LIN {X 0,Y 408.021,Z 164.665,A -85,B 0,C 180,E1 -11041.457,E2 -11041.457} C_VEL
LIN {X 0,Y 408.969,Z 167.841,A -85,B 0,C 180,E1 -11041.957,E2 -11041.957} C_VEL
LIN {X 0,Y 417.373,Z 186.722,A -85,B 0,C 180,E1 -11042.944,E2 -11042.944} C_VEL
LIN {X 0,Y 418.516,Z 191.213,A -85,B 0,C 180,E1 -11043.111,E2 -11043.111} C_VEL
LIN {X 0,Y 416.527,Z 295.761,A -85,B 0,C 180,E1 -11044.949,E2 -11044.949} C_VEL
LIN {X 0,Y 415.758,Z 335.441,A -85,B 0,C 180,E1 -11045.676,E2 -11045.676} C_VEL
LIN {X 0,Y 415.307,Z 350.191,A -85,B 0,C 180,E1 -11046.129,E2 -11046.129} C_VEL
LIN {X 0,Y 414.66,Z 364.218,A -85,B 0,C 180,E1 -11046.741,E2 -11046.741} C_VEL
LIN {X 0,Y 414.075,Z 373.718,A -85,B 0,C 180,E1 -11047.26,E2 -11047.26} C_VEL
LIN {X 0,Y 413.146,Z 379.141,A -85,B 0,C 180,E1 -11047.557,E2 -11047.557} C_VEL
LIN {X 0,Y 409.846,Z 387.886,A -85,B 0,C 180,E1 -11048.015,E2 -11048.015} C_VEL
LIN {X 0,Y 406.373,Z 396.437,A -85,B 0,C 180,E1 -11048.54,E2 -11048.54} C_VEL
LIN {X 0,Y 405.151,Z 401.412,A -85,B 0,C 180,E1 -11048.948,E2 -11048.948} C_VEL
LIN {X 0,Y 403.781,Z 413.481,A -85,B 0,C 180,E1 -11050.194,E2 -11050.194} C_VEL
LIN {X 0,Y 402.539,Z 425.332,A -85,B 0,C 180,E1 -11051.682,E2 -11051.682} C_VEL
LIN {X 0,Y 401.227,Z 435.48,A -85,B 0,C 180,E1 -11053.2,E2 -11053.2} C_VEL
LIN {X 0,Y 399.908,Z 445.382,A -85,B 0,C 180,E1 -11054.975,E2 -11054.975} C_VEL
LIN {X 0,Y 398.903,Z 453.589,A -85,B 0,C 180,E1 -11056.758,E2 -11056.758} C_VEL
LIN {X 0,Y 397.976,Z 461.263,A -85,B 0,C 180,E1 -11058.798,E2 -11058.798} C_VEL
LIN {X 0,Y 397.275,Z 467.361,A -85,B 0,C 180,E1 -11060.837,E2 -11060.837} C_VEL
LIN {X 0,Y 396.768,Z 472.074,A -85,B 0,C 180,E1 -11062.876,E2 -11062.876} C_VEL
LIN {X 0,Y 396.541,Z 475.518,A -85,B 0,C 180,E1 -11064.915,E2 -11064.915} C_VEL
LIN {X 0,Y 396.369,Z 477.793,A -85,B 0,C 180,E1 -11066.95,E2 -11066.95} C_VEL
LIN {X 0,Y 396.082,Z 478.967,A -85,B 0,C 180,E1 -11068.982,E2 -11068.982} C_VEL
LIN {X 0,Y 396.081,Z 478.981,A -85,B 0,C 180,E1 -11071.015,E2 -11071.015} C_VEL
LIN {X 0,Y 396.367,Z 477.865,A -85,B 0,C 180,E1 -11073.048,E2 -11073.048} C_VEL
LIN {X 0,Y 396.529,Z 475.652,A -85,B 0,C 180,E1 -11075.083,E2 -11075.083} C_VEL
LIN {X 0,Y 396.764,Z 472.277,A -85,B 0,C 180,E1 -11077.121,E2 -11077.121} C_VEL
LIN {X 0,Y 397.269,Z 467.633,A -85,B 0,C 180,E1 -11079.16,E2 -11079.16} C_VEL
LIN {X 0,Y 397.952,Z 461.602,A -85,B 0,C 180,E1 -11081.2,E2 -11081.2} C_VEL
LIN {X 0,Y 398.867,Z 454.005,A -85,B 0,C 180,E1 -11083.24,E2 -11083.24} C_VEL
LIN {X 0,Y 399.845,Z 445.978,A -85,B 0,C 180,E1 -11085.008,E2 -11085.008} C_VEL
LIN {X 0,Y 401.166,Z 436.091,A -85,B 0,C 180,E1 -11086.8,E2 -11086.8} C_VEL
LIN {X 0,Y 402.459,Z 426.066,A -85,B 0,C 180,E1 -11088.319,E2 -11088.319} C_VEL
LIN {X 0,Y 403.698,Z 414.655,A -85,B 0,C 180,E1 -11089.773,E2 -11089.773} C_VEL
LIN {X 0,Y 405.129,Z 402.003,A -85,B 0,C 180,E1 -11091.096,E2 -11091.096} C_VEL
LIN {X 0,Y 406.489,Z 388.828,A -85,B 0,C 180,E1 -11092.221,E2 -11092.221} C_VEL
LIN {X 0,Y 407.563,Z 375.261,A -85,B 0,C 180,E1 -11093.163,E2 -11093.163} C_VEL
LIN {X 0,Y 408.376,Z 361.756,A -85,B 0,C 180,E1 -11093.904,E2 -11093.904} C_VEL
LIN {X 0,Y 409.06,Z 346.686,A -85,B 0,C 180,E1 -11094.519,E2 -11094.519} C_VEL
LIN {X 0,Y 409.496,Z 331.535,A -85,B 0,C 180,E1 -11094.931,E2 -11094.931} C_VEL
LIN {X 0,Y 412.244,Z 193.174,A -85,B 0,C 180,E1 -11097.405,E2 -11097.405} C_VEL
LIN {X 0,Y 411.218,Z 189.005,A -85,B 0,C 180,E1 -11097.561,E2 -11097.561} C_VEL
LIN {X 0,Y 402.554,Z 169.768,A -85,B 0,C 180,E1 -11098.604,E2 -11098.604} C_VEL
LIN {X 0,Y 401.881,Z 168.212,A -85,B 0,C 180,E1 -11098.709,E2 -11098.709} C_VEL
LIN {X 0,Y 397.118,Z 152.67,A -85,B 0,C 180,E1 -11101.396,E2 -11101.396} C_VEL
LIN {X 0,Y 397.121,Z 152.643,A -85,B 0,C 180,E1 -11104.492,E2 -11104.492} C_VEL
LIN {X 0,Y 397.098,Z 152.644,A -85,B 0,C 180,E1 -11108.273,E2 -11108.273} C_VEL
LIN {X 0,Y 397.085,Z 152.629,A -85,B 0,C 180,E1 -11110.907,E2 -11110.907} C_VEL
LIN {X 0,Y 397.098,Z 152.641,A -85,B 0,C 180,E1 -11113.647,E2 -11113.647} C_VEL
LIN {X 0,Y 397.097,Z 152.645,A -85,B 0,C 180,E1 -11116.519,E2 -11116.519} C_VEL
LIN {X 0,Y 397.113,Z 152.644,A -85,B 0,C 180,E1 -11119.55,E2 -11119.55} C_VEL
LIN {X 0,Y 397.091,Z 152.645,A -85,B 0,C 180,E1 -11122.789,E2 -11122.789} C_VEL
LIN {X 0,Y 397.11,Z 152.637,A -85,B 0,C 180,E1 -11126.281,E2 -11126.281} C_VEL
LIN {X 0,Y 397.079,Z 152.64,A -85,B 0,C 180,E1 -11129.117,E2 -11129.117} C_VEL
LIN {X 0,Y 397.185,Z 152.635,A -85,B 0,C 180,E1 -11132.609,E2 -11132.609} C_VEL
LIN {X 0,Y 397.119,Z 152.633,A -85,B 0,C 180,E1 -11135.981,E2 -11135.981} C_VEL
LIN {X 0,Y 397.128,Z 152.633,A -85,B 0,C 180,E1 -11139.704,E2 -11139.704} C_VEL
LIN {X 0,Y 397.171,Z 152.633,A -85,B 0,C 180,E1 -11142.844,E2 -11142.844} C_VEL
LIN {X 0,Y 397.215,Z 152.617,A -85,B 0,C 180,E1 -11146.678,E2 -11146.678} C_VEL
LIN {X 0,Y 397.208,Z 152.629,A -85,B 0,C 180,E1 -11149.809,E2 -11149.809} C_VEL
LIN {X 0,Y 397.353,Z 152.598,A -85,B 0,C 180,E1 -11152.888,E2 -11152.888} C_VEL
LIN {X 0,Y 397.245,Z 152.619,A -85,B 0,C 180,E1 -11154.925,E2 -11154.925} C_VEL
LIN {X 0,Y 397.441,Z 152.6,A -85,B 0,C 180,E1 -11157.973,E2 -11157.973} C_VEL
LIN {X 0,Y 397.571,Z 152.569,A -85,B 0,C 180,E1 -11160,E2 -11160} C_VEL
LIN {X 0,Y 397.372,Z 152.611,A -85,B 0,C 180,E1 -11163.041,E2 -11163.041} C_VEL
LIN {X 0,Y 397.352,Z 152.597,A -85,B 0,C 180,E1 -11167.112,E2 -11167.112} C_VEL
LIN {X 0,Y 397.208,Z 152.629,A -85,B 0,C 180,E1 -11170.191,E2 -11170.191} C_VEL
LIN {X 0,Y 397.215,Z 152.613,A -85,B 0,C 180,E1 -11173.321,E2 -11173.321} C_VEL
LIN {X 0,Y 397.16,Z 152.637,A -85,B 0,C 180,E1 -11176.447,E2 -11176.447} C_VEL
LIN {X 0,Y 397.137,Z 152.625,A -85,B 0,C 180,E1 -11179.648,E2 -11179.648} C_VEL
LIN {X 0,Y 397.125,Z 152.635,A -85,B 0,C 180,E1 -11183.041,E2 -11183.041} C_VEL
LIN {X 0,Y 397.125,Z 152.639,A -85,B 0,C 180,E1 -11186.259,E2 -11186.259} C_VEL
LIN {X 0,Y 397.111,Z 152.637,A -85,B 0,C 180,E1 -11188.544,E2 -11188.544} C_VEL
LIN {X 0,Y 397.069,Z 152.651,A -85,B 0,C 180,E1 -11192.072,E2 -11192.072} C_VEL
LIN {X 0,Y 397.11,Z 152.64,A -85,B 0,C 180,E1 -11195.504,E2 -11195.504} C_VEL
LIN {X 0,Y 397.123,Z 152.623,A -85,B 0,C 180,E1 -11198.863,E2 -11198.863} C_VEL
LIN {X 0,Y 397.059,Z 152.636,A -85,B 0,C 180,E1 -11202.268,E2 -11202.268} C_VEL
LIN {X 0,Y 397.109,Z 152.643,A -85,B 0,C 180,E1 -11205.065,E2 -11205.065} C_VEL
LIN {X 0,Y 397.149,Z 152.642,A -85,B 0,C 180,E1 -11208.008,E2 -11208.008} C_VEL
LIN {X 0,Y 397.135,Z 152.637,A -85,B 0,C 180,E1 -11211.989,E2 -11211.989} C_VEL
LIN {X 0,Y 403.812,Z 174.916,A -85,B 0,C 180,E1 -11215.514,E2 -11215.514} C_VEL
LIN {X 0,Y 408.122,Z 189.921,A -85,B 0,C 180,E1 -11217.737,E2 -11217.737} C_VEL
LIN {X 0,Y 405.393,Z 216.791,A -85,B 0,C 180,E1 -11220.962,E2 -11220.962} C_VEL
LIN {X 0,Y 404.786,Z 223.542,A -85,B 0,C 180,E1 -11221.752,E2 -11221.752} C_VEL
LIN {X 0,Y 410.254,Z 268.107,A -85,B 0,C 180,E1 -11223.009,E2 -11223.009} C_VEL
LIN {X 0,Y 408.286,Z 377.569,A -85,B 0,C 180,E1 -11224.956,E2 -11224.956} C_VEL
LIN {X 0,Y 407.723,Z 400.403,A -85,B 0,C 180,E1 -11225.395,E2 -11225.395} C_VEL
LIN {X 0,Y 406.837,Z 415.914,A -85,B 0,C 180,E1 -11225.881,E2 -11225.881} C_VEL
LIN {X 0,Y 405.754,Z 430.277,A -85,B 0,C 180,E1 -11226.525,E2 -11226.525} C_VEL
LIN {X 0,Y 404.634,Z 443.502,A -85,B 0,C 180,E1 -11227.304,E2 -11227.304} C_VEL
LIN {X 0,Y 403.02,Z 458.122,A -85,B 0,C 180,E1 -11228.386,E2 -11228.386} C_VEL
LIN {X 0,Y 401.573,Z 471.663,A -85,B 0,C 180,E1 -11229.647,E2 -11229.647} C_VEL
LIN {X 0,Y 400.174,Z 483.977,A -85,B 0,C 180,E1 -11231.042,E2 -11231.042} C_VEL
LIN {X 0,Y 398.967,Z 495.231,A -85,B 0,C 180,E1 -11232.576,E2 -11232.576} C_VEL
LIN {X 0,Y 397.956,Z 504.72,A -85,B 0,C 180,E1 -11234.115,E2 -11234.115} C_VEL
LIN {X 0,Y 397.129,Z 514.055,A -85,B 0,C 180,E1 -11235.918,E2 -11235.918} C_VEL
LIN {X 0,Y 396.519,Z 521.815,A -85,B 0,C 180,E1 -11237.721,E2 -11237.721} C_VEL
LIN {X 0,Y 396.257,Z 527.426,A -85,B 0,C 180,E1 -11239.269,E2 -11239.269} C_VEL
LIN {X 0,Y 396.049,Z 533.524,A -85,B 0,C 180,E1 -11241.326,E2 -11241.326} C_VEL
LIN {X 0,Y 396.1,Z 538.462,A -85,B 0,C 180,E1 -11243.517,E2 -11243.517} C_VEL
LIN {X 0,Y 396.103,Z 540.808,A -85,B 0,C 180,E1 -11244.912,E2 -11244.912} C_VEL
LIN {X 0,Y 396.218,Z 543.231,A -85,B 0,C 180,E1 -11246.951,E2 -11246.951} C_VEL
LIN {X 0,Y 396.217,Z 544.445,A -85,B 0,C 180,E1 -11248.985,E2 -11248.985} C_VEL
LIN {X 0,Y 396.204,Z 544.443,A -85,B 0,C 180,E1 -11251.018,E2 -11251.018} C_VEL
LIN {X 0,Y 396.219,Z 543.229,A -85,B 0,C 180,E1 -11253.052,E2 -11253.052} C_VEL
LIN {X 0,Y 396.098,Z 540.8,A -85,B 0,C 180,E1 -11255.091,E2 -11255.091} C_VEL
LIN {X 0,Y 396.093,Z 537.12,A -85,B 0,C 180,E1 -11257.136,E2 -11257.136} C_VEL
LIN {X 0,Y 396.105,Z 532.099,A -85,B 0,C 180,E1 -11259.19,E2 -11259.19} C_VEL
LIN {X 0,Y 396.378,Z 525.628,A -85,B 0,C 180,E1 -11261.248,E2 -11261.248} C_VEL
LIN {X 0,Y 396.876,Z 517.511,A -85,B 0,C 180,E1 -11263.31,E2 -11263.31} C_VEL
LIN {X 0,Y 397.589,Z 508.865,A -85,B 0,C 180,E1 -11265.115,E2 -11265.115} C_VEL
LIN {X 0,Y 398.671,Z 498.474,A -85,B 0,C 180,E1 -11266.911,E2 -11266.911} C_VEL
LIN {X 0,Y 399.779,Z 487.843,A -85,B 0,C 180,E1 -11268.449,E2 -11268.449} C_VEL
LIN {X 0,Y 401.029,Z 476.284,A -85,B 0,C 180,E1 -11269.85,E2 -11269.85} C_VEL
LIN {X 0,Y 402.443,Z 463.734,A -85,B 0,C 180,E1 -11271.112,E2 -11271.112} C_VEL
LIN {X 0,Y 403.793,Z 451.687,A -85,B 0,C 180,E1 -11272.111,E2 -11272.111} C_VEL
LIN {X 0,Y 405.091,Z 437.85,A -85,B 0,C 180,E1 -11273.043,E2 -11273.043} C_VEL
LIN {X 0,Y 406.35,Z 422.379,A -85,B 0,C 180,E1 -11273.847,E2 -11273.847} C_VEL
LIN {X 0,Y 407.447,Z 406.722,A -85,B 0,C 180,E1 -11274.422,E2 -11274.422} C_VEL
LIN {X 0,Y 407.975,Z 391.263,A -85,B 0,C 180,E1 -11274.795,E2 -11274.795} C_VEL
LIN {X 0,Y 409.35,Z 324.517,A -85,B 0,C 180,E1 -11275.999,E2 -11275.999} C_VEL
LIN {X 0,Y 411.902,Z 267.787,A -85,B 0,C 180,E1 -11277.413,E2 -11277.413} C_VEL
LIN {X 0,Y 410.199,Z 247.528,A -85,B 0,C 180,E1 -11278.216,E2 -11278.216} C_VEL
LIN {X 0,Y 408.178,Z 233.394,A -85,B 0,C 180,E1 -11278.894,E2 -11278.894} C_VEL
LIN {X 0,Y 412.028,Z 211.405,A -85,B 0,C 180,E1 -11281.923,E2 -11281.923} C_VEL
LIN {X 0,Y 414.392,Z 200.57,A -85,B 0,C 180,E1 -11283.492,E2 -11283.492} C_VEL
LIN {X 0,Y 414.398,Z 198.896,A -85,B 0,C 180,E1 -11283.797,E2 -11283.797} C_VEL
LIN {X 0,Y 412.326,Z 190.433,A -85,B 0,C 180,E1 -11285.794,E2 -11285.794} C_VEL
LIN {X 0,Y 409.948,Z 183.181,A -85,B 0,C 180,E1 -11287.945,E2 -11287.945} C_VEL
LIN {X 0,Y 408.411,Z 178.732,A -85,B 0,C 180,E1 -11289.548,E2 -11289.548} C_VEL
LIN {X 0,Y 407.187,Z 175.487,A -85,B 0,C 180,E1 -11290.987,E2 -11290.987} C_VEL
LIN {X 0,Y 405.558,Z 171.699,A -85,B 0,C 180,E1 -11293.296,E2 -11293.296} C_VEL
LIN {X 0,Y 404.597,Z 169.529,A -85,B 0,C 180,E1 -11295.414,E2 -11295.414} C_VEL
LIN {X 0,Y 404.292,Z 168.538,A -85,B 0,C 180,E1 -11297.316,E2 -11297.316} C_VEL
LIN {X 0,Y 404.141,Z 168.532,A -85,B 0,C 180,E1 -11298.638,E2 -11298.638} C_VEL
LIN {X 0,Y 404.304,Z 169.873,A -85,B 0,C 180,E1 -11301.26,E2 -11301.26} C_VEL
LIN {X 0,Y 405.298,Z 172.634,A -85,B 0,C 180,E1 -11303.874,E2 -11303.874} C_VEL
LIN {X 0,Y 406.441,Z 176.266,A -85,B 0,C 180,E1 -11306.1,E2 -11306.1} C_VEL
LIN {X 0,Y 407.654,Z 180.67,A -85,B 0,C 180,E1 -11308.189,E2 -11308.189} C_VEL
LIN {X 0,Y 409.124,Z 187.192,A -85,B 0,C 180,E1 -11310.688,E2 -11310.688} C_VEL
LIN {X 0,Y 410.116,Z 192.489,A -85,B 0,C 180,E1 -11312.439,E2 -11312.439} C_VEL
LIN {X 0,Y 410.527,Z 196.337,A -85,B 0,C 180,E1 -11313.57,E2 -11313.57} C_VEL
LIN {X 0,Y 408.558,Z 207.239,A -85,B 0,C 180,E1 -11316.061,E2 -11316.061} C_VEL
LIN {X 0,Y 408.206,Z 209.863,A -85,B 0,C 180,E1 -11316.608,E2 -11316.608} C_VEL
LIN {X 0,Y 412.045,Z 224.419,A -85,B 0,C 180,E1 -11317.661,E2 -11317.661} C_VEL
LIN {X 0,Y 413.131,Z 229.704,A -85,B 0,C 180,E1 -11317.992,E2 -11317.992} C_VEL
LIN {X 0,Y 407.346,Z 316.237,A -85,B 0,C 180,E1 -11320.668,E2 -11320.668} C_VEL
LIN {X 0,Y 406.778,Z 332.313,A -85,B 0,C 180,E1 -11321.229,E2 -11321.229} C_VEL
LIN {X 0,Y 406.107,Z 346.202,A -85,B 0,C 180,E1 -11321.914,E2 -11321.914} C_VEL
LIN {X 0,Y 405.155,Z 360.459,A -85,B 0,C 180,E1 -11322.849,E2 -11322.849} C_VEL
LIN {X 0,Y 404.107,Z 373.535,A -85,B 0,C 180,E1 -11323.973,E2 -11323.973} C_VEL
LIN {X 0,Y 403.231,Z 384.092,A -85,B 0,C 180,E1 -11325.103,E2 -11325.103} C_VEL
LIN {X 0,Y 402.315,Z 393.688,A -85,B 0,C 180,E1 -11326.36,E2 -11326.36} C_VEL
LIN {X 0,Y 401.261,Z 403.094,A -85,B 0,C 180,E1 -11327.867,E2 -11327.867} C_VEL
LIN {X 0,Y 400.302,Z 411.148,A -85,B 0,C 180,E1 -11329.48,E2 -11329.48} C_VEL
LIN {X 0,Y 399.468,Z 416.812,A -85,B 0,C 180,E1 -11330.89,E2 -11330.89} C_VEL
LIN {X 0,Y 398.948,Z 421.58,A -85,B 0,C 180,E1 -11332.408,E2 -11332.408} C_VEL
LIN {X 0,Y 398.318,Z 425.26,A -85,B 0,C 180,E1 -11333.923,E2 -11333.923} C_VEL
LIN {X 0,Y 398.058,Z 427.078,A -85,B 0,C 180,E1 -11334.936,E2 -11334.936} C_VEL
LIN {X 0,Y 397.873,Z 428.461,A -85,B 0,C 180,E1 -11335.948,E2 -11335.948} C_VEL
LIN {X 0,Y 397.665,Z 429.44,A -85,B 0,C 180,E1 -11336.961,E2 -11336.961} C_VEL
LIN {X 0,Y 397.525,Z 429.977,A -85,B 0,C 180,E1 -11337.974,E2 -11337.974} C_VEL
LIN {X 0,Y 397.299,Z 430.089,A -85,B 0,C 180,E1 -11338.987,E2 -11338.987} C_VEL
LIN {X 0,Y 397.206,Z 429.774,A -85,B 0,C 180,E1 -11340,E2 -11340} C_VEL
LIN {X 0,Y 397.219,Z 429.042,A -85,B 0,C 180,E1 -11341.014,E2 -11341.014} C_VEL
LIN {X 0,Y 397.141,Z 427.889,A -85,B 0,C 180,E1 -11342.028,E2 -11342.028} C_VEL
LIN {X 0,Y 397.147,Z 425.347,A -85,B 0,C 180,E1 -11343.551,E2 -11343.551} C_VEL
LIN {X 0,Y 397.263,Z 421.771,A -85,B 0,C 180,E1 -11345.075,E2 -11345.075} C_VEL
LIN {X 0,Y 397.527,Z 417.087,A -85,B 0,C 180,E1 -11346.599,E2 -11346.599} C_VEL
LIN {X 0,Y 397.823,Z 411.176,A -85,B 0,C 180,E1 -11348.125,E2 -11348.125} C_VEL
LIN {X 0,Y 398.204,Z 403.848,A -85,B 0,C 180,E1 -11349.652,E2 -11349.652} C_VEL
LIN {X 0,Y 398.702,Z 394.845,A -85,B 0,C 180,E1 -11351.181,E2 -11351.181} C_VEL
LIN {X 0,Y 399.232,Z 384.652,A -85,B 0,C 180,E1 -11352.583,E2 -11352.583} C_VEL
LIN {X 0,Y 399.846,Z 373.252,A -85,B 0,C 180,E1 -11353.856,E2 -11353.856} C_VEL
LIN {X 0,Y 400.359,Z 361.658,A -85,B 0,C 180,E1 -11354.907,E2 -11354.907} C_VEL
LIN {X 0,Y 400.866,Z 348.717,A -85,B 0,C 180,E1 -11355.834,E2 -11355.834} C_VEL
LIN {X 0,Y 401.238,Z 336.062,A -85,B 0,C 180,E1 -11356.537,E2 -11356.537} C_VEL
LIN {X 0,Y 401.582,Z 323.646,A -85,B 0,C 180,E1 -11357.046,E2 -11357.046} C_VEL
LIN {X 0,Y 401.849,Z 305.487,A -85,B 0,C 180,E1 -11357.526,E2 -11357.526} C_VEL
LIN {X 0,Y 403.894,Z 221.695,A -85,B 0,C 180,E1 -11359.463,E2 -11359.463} C_VEL
LIN {X 0,Y 400.491,Z 201.256,A -85,B 0,C 180,E1 -11360.141,E2 -11360.141} C_VEL
LIN {X 0,Y 401.81,Z 182.13,A -85,B 0,C 180,E1 -11363.722,E2 -11363.722} C_VEL
LIN {X 0,Y 402.035,Z 175.04,A -85,B 0,C 180,E1 -11365.082,E2 -11365.082} C_VEL
LIN {X 0,Y 399.379,Z 162.271,A -85,B 0,C 180,E1 -11367.757,E2 -11367.757} C_VEL
LIN {X 0,Y 397.107,Z 152.647,A -85,B 0,C 180,E1 -11369.863,E2 -11369.863} C_VEL
LIN {X 0,Y 397.124,Z 152.644,A -85,B 0,C 180,E1 -11373.717,E2 -11373.717} C_VEL
LIN {X 0,Y 397.097,Z 152.648,A -85,B 0,C 180,E1 -11377.208,E2 -11377.208} C_VEL
LIN {X 0,Y 397.082,Z 152.639,A -85,B 0,C 180,E1 -11380.441,E2 -11380.441} C_VEL
LIN {X 0,Y 397.105,Z 152.637,A -85,B 0,C 180,E1 -11383.648,E2 -11383.648} C_VEL
LIN {X 0,Y 397.107,Z 152.643,A -85,B 0,C 180,E1 -11386.52,E2 -11386.52} C_VEL
LIN {X 0,Y 397.118,Z 152.639,A -85,B 0,C 180,E1 -11390.422,E2 -11390.422} C_VEL
LIN {X 0,Y 397.112,Z 152.649,A -85,B 0,C 180,E1 -11394.265,E2 -11394.265} C_VEL
LIN {X 0,Y 397.119,Z 152.644,A -85,B 0,C 180,E1 -11396.726,E2 -11396.726} C_VEL
LIN {X 0,Y 397.125,Z 152.734,A -85,B 0,C 180,E1 -11398.713,E2 -11398.713} C_VEL
LIN {X 0,Y 401.677,Z 167.617,A -85,B 0,C 180,E1 -11401.3,E2 -11401.3} C_VEL
LIN {X 0,Y 401.981,Z 168.544,A -85,B 0,C 180,E1 -11401.429,E2 -11401.429} C_VEL
LIN {X 0,Y 410.806,Z 187.932,A -85,B 0,C 180,E1 -11402.488,E2 -11402.488} C_VEL
LIN {X 0,Y 412.127,Z 192.143,A -85,B 0,C 180,E1 -11402.668,E2 -11402.668} C_VEL
LIN {X 0,Y 410.317,Z 287.367,A -85,B 0,C 180,E1 -11404.373,E2 -11404.373} C_VEL
LIN {X 0,Y 409.324,Z 335.96,A -85,B 0,C 180,E1 -11405.268,E2 -11405.268} C_VEL
LIN {X 0,Y 408.852,Z 350.887,A -85,B 0,C 180,E1 -11405.734,E2 -11405.734} C_VEL
LIN {X 0,Y 408.173,Z 364.968,A -85,B 0,C 180,E1 -11406.36,E2 -11406.36} C_VEL
LIN {X 0,Y 407.292,Z 378.606,A -85,B 0,C 180,E1 -11407.153,E2 -11407.153} C_VEL
LIN {X 0,Y 406.113,Z 392.307,A -85,B 0,C 180,E1 -11408.156,E2 -11408.156} C_VEL
LIN {X 0,Y 405.151,Z 401.412,A -85,B 0,C 180,E1 -11408.948,E2 -11408.948} C_VEL
LIN {X 0,Y 403.955,Z 406.344,A -85,B 0,C 180,E1 -11409.378,E2 -11409.378} C_VEL
LIN {X 0,Y 400.447,Z 414.245,A -85,B 0,C 180,E1 -11410.068,E2 -11410.068} C_VEL
LIN {X 0,Y 396.954,Z 421.797,A -85,B 0,C 180,E1 -11410.839,E2 -11410.839} C_VEL
LIN {X 0,Y 395.793,Z 426.121,A -85,B 0,C 180,E1 -11411.389,E2 -11411.389} C_VEL
LIN {X 0,Y 394.451,Z 436.062,A -85,B 0,C 180,E1 -11412.902,E2 -11412.902} C_VEL
LIN {X 0,Y 393.089,Z 445.755,A -85,B 0,C 180,E1 -11414.665,E2 -11414.665} C_VEL
LIN {X 0,Y 392.014,Z 454.174,A -85,B 0,C 180,E1 -11416.521,E2 -11416.521} C_VEL
LIN {X 0,Y 391.009,Z 461.85,A -85,B 0,C 180,E1 -11418.595,E2 -11418.595} C_VEL
LIN {X 0,Y 390.274,Z 467.948,A -85,B 0,C 180,E1 -11420.672,E2 -11420.672} C_VEL
LIN {X 0,Y 389.748,Z 472.659,A -85,B 0,C 180,E1 -11422.747,E2 -11422.747} C_VEL
LIN {X 0,Y 389.485,Z 476.104,A -85,B 0,C 180,E1 -11424.822,E2 -11424.822} C_VEL
LIN {X 0,Y 389.298,Z 478.379,A -85,B 0,C 180,E1 -11426.894,E2 -11426.894} C_VEL
LIN {X 0,Y 389.031,Z 479.55,A -85,B 0,C 180,E1 -11428.964,E2 -11428.964} C_VEL
LIN {X 0,Y 389.03,Z 479.564,A -85,B 0,C 180,E1 -11431.034,E2 -11431.034} C_VEL
LIN {X 0,Y 389.296,Z 478.45,A -85,B 0,C 180,E1 -11433.103,E2 -11433.103} C_VEL
LIN {X 0,Y 389.473,Z 476.237,A -85,B 0,C 180,E1 -11435.175,E2 -11435.175} C_VEL
LIN {X 0,Y 389.804,Z 472.524,A -85,B 0,C 180,E1 -11437.419,E2 -11437.419} C_VEL
LIN {X 0,Y 390.267,Z 468.217,A -85,B 0,C 180,E1 -11439.326,E2 -11439.326} C_VEL
LIN {X 0,Y 390.982,Z 462.186,A -85,B 0,C 180,E1 -11441.403,E2 -11441.403} C_VEL
LIN {X 0,Y 391.979,Z 454.585,A -85,B 0,C 180,E1 -11443.477,E2 -11443.477} C_VEL
LIN {X 0,Y 393,Z 446.678,A -85,B 0,C 180,E1 -11445.251,E2 -11445.251} C_VEL
LIN {X 0,Y 394.183,Z 438.211,A -85,B 0,C 180,E1 -11446.84,E2 -11446.84} C_VEL
LIN {X 0,Y 395.503,Z 428.421,A -85,B 0,C 180,E1 -11448.384,E2 -11448.384} C_VEL
LIN {X 0,Y 396.863,Z 417.195,A -85,B 0,C 180,E1 -11449.876,E2 -11449.876} C_VEL
LIN {X 0,Y 398.228,Z 405.136,A -85,B 0,C 180,E1 -11451.208,E2 -11451.208} C_VEL
LIN {X 0,Y 399.617,Z 392.51,A -85,B 0,C 180,E1 -11452.352,E2 -11452.352} C_VEL
LIN {X 0,Y 400.802,Z 378.716,A -85,B 0,C 180,E1 -11453.372,E2 -11453.372} C_VEL
LIN {X 0,Y 401.83,Z 364.343,A -85,B 0,C 180,E1 -11454.204,E2 -11454.204} C_VEL
LIN {X 0,Y 402.491,Z 349.785,A -85,B 0,C 180,E1 -11454.843,E2 -11454.843} C_VEL
LIN {X 0,Y 402.995,Z 334.732,A -85,B 0,C 180,E1 -11455.293,E2 -11455.293} C_VEL
LIN {X 0,Y 405.875,Z 198.835,A -85,B 0,C 180,E1 -11457.769,E2 -11457.769} C_VEL
LIN {X 0,Y 405.868,Z 193.622,A -85,B 0,C 180,E1 -11457.872,E2 -11457.872} C_VEL
LIN {X 0,Y 400.034,Z 179.778,A -85,B 0,C 180,E1 -11458.603,E2 -11458.603} C_VEL
LIN {X 0,Y 394.796,Z 168.752,A -85,B 0,C 180,E1 -11459.275,E2 -11459.275} C_VEL
LIN {X 0,Y 390.908,Z 156.366,A -85,B 0,C 180,E1 -11461.423,E2 -11461.423} C_VEL
LIN {X 0,Y 390.04,Z 153.515,A -85,B 0,C 180,E1 -11461.987,E2 -11461.987} C_VEL
LIN {X 0,Y 390.081,Z 153.521,A -85,B 0,C 180,E1 -11465.205,E2 -11465.205} C_VEL
LIN {X 0,Y 390.084,Z 153.505,A -85,B 0,C 180,E1 -11469.091,E2 -11469.091} C_VEL
LIN {X 0,Y 390.057,Z 153.522,A -85,B 0,C 180,E1 -11472.376,E2 -11472.376} C_VEL
LIN {X 0,Y 390.048,Z 153.523,A -85,B 0,C 180,E1 -11476.112,E2 -11476.112} C_VEL
LIN {X 0,Y 390.067,Z 153.521,A -85,B 0,C 180,E1 -11479.562,E2 -11479.562} C_VEL
LIN {X 0,Y 390.039,Z 153.521,A -85,B 0,C 180,E1 -11482.447,E2 -11482.447} C_VEL
LIN {X 0,Y 390.075,Z 153.514,A -85,B 0,C 180,E1 -11486.046,E2 -11486.046} C_VEL
LIN {X 0,Y 390.036,Z 153.511,A -85,B 0,C 180,E1 -11489.7,E2 -11489.7} C_VEL
LIN {X 0,Y 390.104,Z 153.516,A -85,B 0,C 180,E1 -11493.231,E2 -11493.231} C_VEL
LIN {X 0,Y 390.066,Z 153.516,A -85,B 0,C 180,E1 -11496.76,E2 -11496.76} C_VEL
LIN {X 0,Y 390.093,Z 153.509,A -85,B 0,C 180,E1 -11499.982,E2 -11499.982} C_VEL
LIN {X 0,Y 390.127,Z 153.515,A -85,B 0,C 180,E1 -11503.248,E2 -11503.248} C_VEL
LIN {X 0,Y 390.183,Z 153.494,A -85,B 0,C 180,E1 -11506.561,E2 -11506.561} C_VEL
LIN {X 0,Y 390.159,Z 153.508,A -85,B 0,C 180,E1 -11509.622,E2 -11509.622} C_VEL
LIN {X 0,Y 390.307,Z 153.477,A -85,B 0,C 180,E1 -11512.759,E2 -11512.759} C_VEL
LIN {X 0,Y 390.217,Z 153.492,A -85,B 0,C 180,E1 -11514.833,E2 -11514.833} C_VEL
LIN {X 0,Y 390.41,Z 153.476,A -85,B 0,C 180,E1 -11517.937,E2 -11517.937} C_VEL
LIN {X 0,Y 390.541,Z 153.444,A -85,B 0,C 180,E1 -11520,E2 -11520} C_VEL
LIN {X 0,Y 390.306,Z 153.49,A -85,B 0,C 180,E1 -11523.096,E2 -11523.096} C_VEL
LIN {X 0,Y 390.319,Z 153.474,A -85,B 0,C 180,E1 -11526.202,E2 -11526.202} C_VEL
LIN {X 0,Y 390.303,Z 153.48,A -85,B 0,C 180,E1 -11528.282,E2 -11528.282} C_VEL
LIN {X 0,Y 390.16,Z 153.493,A -85,B 0,C 180,E1 -11532.483,E2 -11532.483} C_VEL
LIN {X 0,Y 390.133,Z 153.507,A -85,B 0,C 180,E1 -11535.677,E2 -11535.677} C_VEL
LIN {X 0,Y 390.095,Z 153.501,A -85,B 0,C 180,E1 -11538.922,E2 -11538.922} C_VEL
LIN {X 0,Y 390.031,Z 153.527,A -85,B 0,C 180,E1 -11542.235,E2 -11542.235} C_VEL
LIN {X 0,Y 390.108,Z 153.508,A -85,B 0,C 180,E1 -11545.744,E2 -11545.744} C_VEL
LIN {X 0,Y 390.048,Z 153.512,A -85,B 0,C 180,E1 -11549.11,E2 -11549.11} C_VEL
LIN {X 0,Y 390.033,Z 153.523,A -85,B 0,C 180,E1 -11552.722,E2 -11552.722} C_VEL
LIN {X 0,Y 390.048,Z 153.522,A -85,B 0,C 180,E1 -11555.827,E2 -11555.827} C_VEL
LIN {X 0,Y 390.062,Z 153.495,A -85,B 0,C 180,E1 -11559.22,E2 -11559.22} C_VEL
LIN {X 0,Y 390.033,Z 153.513,A -85,B 0,C 180,E1 -11562.375,E2 -11562.375} C_VEL
LIN {X 0,Y 390.098,Z 153.519,A -85,B 0,C 180,E1 -11566.107,E2 -11566.107} C_VEL
LIN {X 0,Y 390.075,Z 153.521,A -85,B 0,C 180,E1 -11569.175,E2 -11569.175} C_VEL
LIN {X 0,Y 390.093,Z 153.561,A -85,B 0,C 180,E1 -11571.564,E2 -11571.564} C_VEL
LIN {X 0,Y 396.406,Z 174.706,A -85,B 0,C 180,E1 -11574.967,E2 -11574.967} C_VEL
LIN {X 0,Y 401.15,Z 191.216,A -85,B 0,C 180,E1 -11577.472,E2 -11577.472} C_VEL
LIN {X 0,Y 401.189,Z 193.586,A -85,B 0,C 180,E1 -11577.783,E2 -11577.783} C_VEL
LIN {X 0,Y 398.167,Z 221.719,A -85,B 0,C 180,E1 -11581.209,E2 -11581.209} C_VEL
LIN {X 0,Y 403.756,Z 267.493,A -85,B 0,C 180,E1 -11582.535,E2 -11582.535} C_VEL
LIN {X 0,Y 403.807,Z 278.072,A -85,B 0,C 180,E1 -11582.745,E2 -11582.745} C_VEL
LIN {X 0,Y 401.363,Z 397.31,A -85,B 0,C 180,E1 -11584.909,E2 -11584.909} C_VEL
LIN {X 0,Y 400.53,Z 412.93,A -85,B 0,C 180,E1 -11585.373,E2 -11585.373} C_VEL
LIN {X 0,Y 399.435,Z 427.254,A -85,B 0,C 180,E1 -11585.993,E2 -11585.993} C_VEL
LIN {X 0,Y 398.286,Z 439.913,A -85,B 0,C 180,E1 -11586.713,E2 -11586.713} C_VEL
LIN {X 0,Y 396.781,Z 454.415,A -85,B 0,C 180,E1 -11587.754,E2 -11587.754} C_VEL
LIN {X 0,Y 395.296,Z 467.247,A -85,B 0,C 180,E1 -11588.9,E2 -11588.9} C_VEL
LIN {X 0,Y 393.776,Z 480.21,A -85,B 0,C 180,E1 -11590.315,E2 -11590.315} C_VEL
LIN {X 0,Y 392.64,Z 490.715,A -85,B 0,C 180,E1 -11591.694,E2 -11591.694} C_VEL
LIN {X 0,Y 391.439,Z 501.122,A -85,B 0,C 180,E1 -11593.307,E2 -11593.307} C_VEL
LIN {X 0,Y 390.329,Z 510.953,A -85,B 0,C 180,E1 -11595.135,E2 -11595.135} C_VEL
LIN {X 0,Y 389.704,Z 518.751,A -85,B 0,C 180,E1 -11596.867,E2 -11596.867} C_VEL
LIN {X 0,Y 389.212,Z 526.836,A -85,B 0,C 180,E1 -11599.072,E2 -11599.072} C_VEL
LIN {X 0,Y 388.945,Z 532.932,A -85,B 0,C 180,E1 -11601.166,E2 -11601.166} C_VEL
LIN {X 0,Y 389.003,Z 536.551,A -85,B 0,C 180,E1 -11602.736,E2 -11602.736} C_VEL
LIN {X 0,Y 389.029,Z 540.222,A -85,B 0,C 180,E1 -11604.819,E2 -11604.819} C_VEL
LIN {X 0,Y 389.146,Z 542.646,A -85,B 0,C 180,E1 -11606.896,E2 -11606.896} C_VEL
LIN {X 0,Y 389.157,Z 543.861,A -85,B 0,C 180,E1 -11608.967,E2 -11608.967} C_VEL
LIN {X 0,Y 389.145,Z 543.86,A -85,B 0,C 180,E1 -11611.036,E2 -11611.036} C_VEL
LIN {X 0,Y 389.146,Z 542.644,A -85,B 0,C 180,E1 -11613.107,E2 -11613.107} C_VEL
LIN {X 0,Y 389.027,Z 540.213,A -85,B 0,C 180,E1 -11615.184,E2 -11615.184} C_VEL
LIN {X 0,Y 389.088,Z 537.938,A -85,B 0,C 180,E1 -11616.562,E2 -11616.562} C_VEL
LIN {X 0,Y 388.997,Z 532.909,A -85,B 0,C 180,E1 -11618.835,E2 -11618.835} C_VEL
LIN {X 0,Y 389.235,Z 526.809,A -85,B 0,C 180,E1 -11620.93,E2 -11620.93} C_VEL
LIN {X 0,Y 389.707,Z 518.72,A -85,B 0,C 180,E1 -11623.135,E2 -11623.135} C_VEL
LIN {X 0,Y 390.498,Z 509.643,A -85,B 0,C 180,E1 -11625.129,E2 -11625.129} C_VEL
LIN {X 0,Y 391.625,Z 499.532,A -85,B 0,C 180,E1 -11626.956,E2 -11626.956} C_VEL
LIN {X 0,Y 392.835,Z 488.372,A -85,B 0,C 180,E1 -11628.633,E2 -11628.633} C_VEL
LIN {X 0,Y 394.137,Z 476.864,A -85,B 0,C 180,E1 -11630.076,E2 -11630.076} C_VEL
LIN {X 0,Y 395.75,Z 463.151,A -85,B 0,C 180,E1 -11631.487,E2 -11631.487} C_VEL
LIN {X 0,Y 397.356,Z 449.419,A -85,B 0,C 180,E1 -11632.626,E2 -11632.626} C_VEL
LIN {X 0,Y 398.67,Z 436.324,A -85,B 0,C 180,E1 -11633.502,E2 -11633.502} C_VEL
LIN {X 0,Y 399.836,Z 421.818,A -85,B 0,C 180,E1 -11634.261,E2 -11634.261} C_VEL
LIN {X 0,Y 400.997,Z 406.185,A -85,B 0,C 180,E1 -11634.841,E2 -11634.841} C_VEL
LIN {X 0,Y 401.54,Z 390.769,A -85,B 0,C 180,E1 -11635.22,E2 -11635.22} C_VEL
LIN {X 0,Y 402.673,Z 339.959,A -85,B 0,C 180,E1 -11636.15,E2 -11636.15} C_VEL
LIN {X 0,Y 406.129,Z 269.157,A -85,B 0,C 180,E1 -11637.958,E2 -11637.958} C_VEL
LIN {X 0,Y 404.492,Z 248.493,A -85,B 0,C 180,E1 -11638.804,E2 -11638.804} C_VEL
LIN {X 0,Y 402.287,Z 232.876,A -85,B 0,C 180,E1 -11639.61,E2 -11639.61} C_VEL
LIN {X 0,Y 406.525,Z 211.111,A -85,B 0,C 180,E1 -11642.702,E2 -11642.702} C_VEL
LIN {X 0,Y 408.31,Z 203.548,A -85,B 0,C 180,E1 -11643.831,E2 -11643.831} C_VEL
LIN {X 0,Y 408.413,Z 202.297,A -85,B 0,C 180,E1 -11644.049,E2 -11644.049} C_VEL
LIN {X 0,Y 406.576,Z 194.328,A -85,B 0,C 180,E1 -11645.996,E2 -11645.996} C_VEL
LIN {X 0,Y 404.541,Z 187.906,A -85,B 0,C 180,E1 -11647.939,E2 -11647.939} C_VEL
LIN {X 0,Y 402.798,Z 182.766,A -85,B 0,C 180,E1 -11649.852,E2 -11649.852} C_VEL
LIN {X 0,Y 401.323,Z 178.925,A -85,B 0,C 180,E1 -11651.719,E2 -11651.719} C_VEL
LIN {X 0,Y 399.976,Z 175.763,A -85,B 0,C 180,E1 -11653.912,E2 -11653.912} C_VEL
LIN {X 0,Y 399.177,Z 173.799,A -85,B 0,C 180,E1 -11656.209,E2 -11656.209} C_VEL
LIN {X 0,Y 398.918,Z 173.233,A -85,B 0,C 180,E1 -11657.974,E2 -11657.974} C_VEL
LIN {X 0,Y 398.79,Z 173.468,A -85,B 0,C 180,E1 -11659.303,E2 -11659.303} C_VEL
LIN {X 0,Y 399.105,Z 175.107,A -85,B 0,C 180,E1 -11661.952,E2 -11661.952} C_VEL
LIN {X 0,Y 399.853,Z 177.282,A -85,B 0,C 180,E1 -11663.953,E2 -11663.953} C_VEL
LIN {X 0,Y 401.084,Z 181.593,A -85,B 0,C 180,E1 -11666.581,E2 -11666.581} C_VEL
LIN {X 0,Y 402.287,Z 186.595,A -85,B 0,C 180,E1 -11668.876,E2 -11668.876} C_VEL
LIN {X 0,Y 403.649,Z 193.32,A -85,B 0,C 180,E1 -11671.393,E2 -11671.393} C_VEL
LIN {X 0,Y 404.352,Z 198.818,A -85,B 0,C 180,E1 -11673.134,E2 -11673.134} C_VEL
LIN {X 0,Y 403.954,Z 202.002,A -85,B 0,C 180,E1 -11673.941,E2 -11673.941} C_VEL
LIN {X 0,Y 402.277,Z 210.419,A -85,B 0,C 180,E1 -11675.865,E2 -11675.865} C_VEL
LIN {X 0,Y 406.039,Z 224.773,A -85,B 0,C 180,E1 -11676.977,E2 -11676.977} C_VEL
LIN {X 0,Y 407.45,Z 231.619,A -85,B 0,C 180,E1 -11677.432,E2 -11677.432} C_VEL
LIN {X 0,Y 401.233,Z 318.071,A -85,B 0,C 180,E1 -11680.195,E2 -11680.195} C_VEL
LIN {X 0,Y 400.557,Z 334.464,A -85,B 0,C 180,E1 -11680.793,E2 -11680.793} C_VEL
LIN {X 0,Y 399.862,Z 347.878,A -85,B 0,C 180,E1 -11681.49,E2 -11681.49} C_VEL
LIN {X 0,Y 398.82,Z 361.965,A -85,B 0,C 180,E1 -11682.441,E2 -11682.441} C_VEL
LIN {X 0,Y 397.726,Z 374.823,A -85,B 0,C 180,E1 -11683.577,E2 -11683.577} C_VEL
LIN {X 0,Y 396.653,Z 386.357,A -85,B 0,C 180,E1 -11684.85,E2 -11684.85} C_VEL
LIN {X 0,Y 395.684,Z 395.709,A -85,B 0,C 180,E1 -11686.126,E2 -11686.126} C_VEL
LIN {X 0,Y 394.545,Z 404.948,A -85,B 0,C 180,E1 -11687.658,E2 -11687.658} C_VEL
LIN {X 0,Y 393.657,Z 411.941,A -85,B 0,C 180,E1 -11689.093,E2 -11689.093} C_VEL
LIN {X 0,Y 392.631,Z 418.369,A -85,B 0,C 180,E1 -11690.729,E2 -11690.729} C_VEL
LIN {X 0,Y 392.065,Z 423.031,A -85,B 0,C 180,E1 -11692.274,E2 -11692.274} C_VEL
LIN {X 0,Y 391.39,Z 426.621,A -85,B 0,C 180,E1 -11693.815,E2 -11693.815} C_VEL
LIN {X 0,Y 391.108,Z 428.386,A -85,B 0,C 180,E1 -11694.845,E2 -11694.845} C_VEL
LIN {X 0,Y 390.919,Z 429.715,A -85,B 0,C 180,E1 -11695.876,E2 -11695.876} C_VEL
LIN {X 0,Y 390.689,Z 430.646,A -85,B 0,C 180,E1 -11696.907,E2 -11696.907} C_VEL
LIN {X 0,Y 390.529,Z 431.108,A -85,B 0,C 180,E1 -11697.937,E2 -11697.937} C_VEL
LIN {X 0,Y 390.305,Z 431.167,A -85,B 0,C 180,E1 -11698.968,E2 -11698.968} C_VEL
LIN {X 0,Y 390.182,Z 430.805,A -85,B 0,C 180,E1 -11700,E2 -11700} C_VEL
LIN {X 0,Y 390.193,Z 430.018,A -85,B 0,C 180,E1 -11701.032,E2 -11701.032} C_VEL
LIN {X 0,Y 390.118,Z 428.789,A -85,B 0,C 180,E1 -11702.065,E2 -11702.065} C_VEL
LIN {X 0,Y 390.118,Z 426.15,A -85,B 0,C 180,E1 -11703.615,E2 -11703.615} C_VEL
LIN {X 0,Y 390.247,Z 422.474,A -85,B 0,C 180,E1 -11705.166,E2 -11705.166} C_VEL
LIN {X 0,Y 390.517,Z 417.683,A -85,B 0,C 180,E1 -11706.718,E2 -11706.718} C_VEL
LIN {X 0,Y 390.788,Z 411.658,A -85,B 0,C 180,E1 -11708.272,E2 -11708.272} C_VEL
LIN {X 0,Y 391.215,Z 404.2,A -85,B 0,C 180,E1 -11709.827,E2 -11709.827} C_VEL
LIN {X 0,Y 391.735,Z 395.041,A -85,B 0,C 180,E1 -11711.382,E2 -11711.382} C_VEL
LIN {X 0,Y 392.283,Z 384.63,A -85,B 0,C 180,E1 -11712.809,E2 -11712.809} C_VEL
LIN {X 0,Y 392.914,Z 373.027,A -85,B 0,C 180,E1 -11714.106,E2 -11714.106} C_VEL
LIN {X 0,Y 393.434,Z 361.096,A -85,B 0,C 180,E1 -11715.176,E2 -11715.176} C_VEL
LIN {X 0,Y 393.959,Z 347.849,A -85,B 0,C 180,E1 -11716.119,E2 -11716.119} C_VEL
LIN {X 0,Y 394.314,Z 333.883,A -85,B 0,C 180,E1 -11716.869,E2 -11716.869} C_VEL
LIN {X 0,Y 394.741,Z 319.324,A -85,B 0,C 180,E1 -11717.418,E2 -11717.418} C_VEL
LIN {X 0,Y 396.989,Z 221.935,A -85,B 0,C 180,E1 -11719.756,E2 -11719.756} C_VEL
LIN {X 0,Y 393.601,Z 201.497,A -85,B 0,C 180,E1 -11720.453,E2 -11720.453} C_VEL
LIN {X 0,Y 394.931,Z 183.374,A -85,B 0,C 180,E1 -11723.882,E2 -11723.882} C_VEL
LIN {X 0,Y 395.273,Z 177.929,A -85,B 0,C 180,E1 -11724.933,E2 -11724.933} C_VEL
LIN {X 0,Y 393.956,Z 170.487,A -85,B 0,C 180,E1 -11726.487,E2 -11726.487} C_VEL
LIN {X 0,Y 390.952,Z 157.361,A -85,B 0,C 180,E1 -11729.332,E2 -11729.332} C_VEL
LIN {X 0,Y 390.055,Z 153.524,A -85,B 0,C 180,E1 -11730.232,E2 -11730.232} C_VEL
LIN {X 0,Y 390.074,Z 153.521,A -85,B 0,C 180,E1 -11734.024,E2 -11734.024} C_VEL
LIN {X 0,Y 390.046,Z 153.526,A -85,B 0,C 180,E1 -11737.55,E2 -11737.55} C_VEL
LIN {X 0,Y 390.037,Z 153.518,A -85,B 0,C 180,E1 -11740.817,E2 -11740.817} C_VEL
LIN {X 0,Y 390.059,Z 153.514,A -85,B 0,C 180,E1 -11743.885,E2 -11743.885} C_VEL
LIN {X 0,Y 390.062,Z 153.518,A -85,B 0,C 180,E1 -11746.789,E2 -11746.789} C_VEL
LIN {X 0,Y 390.061,Z 153.518,A -85,B 0,C 180,E1 -11749.56,E2 -11749.56} C_VEL
LIN {X 0,Y 390.047,Z 153.524,A -85,B 0,C 180,E1 -11752.449,E2 -11752.449} C_VEL
LIN {X 0,Y 390.073,Z 153.525,A -85,B 0,C 180,E1 -11756.044,E2 -11756.044} C_VEL
LIN {X 0,Y 390.053,Z 153.566,A -85,B 0,C 180,E1 -11758.166,E2 -11758.166} C_VEL
LIN {X 0,Y 394.816,Z 168.798,A -85,B 0,C 180,E1 -11760.839,E2 -11760.839} C_VEL
LIN {X 0,Y 403.106,Z 186.722,A -85,B 0,C 180,E1 -11761.881,E2 -11761.881} C_VEL
LIN {X 0,Y 405.887,Z 193.761,A -85,B 0,C 180,E1 -11762.234,E2 -11762.234} C_VEL
LIN {X 0,Y 403.754,Z 296.75,A -85,B 0,C 180,E1 -11764.099,E2 -11764.099} C_VEL
LIN {X 0,Y 402.876,Z 337.427,A -85,B 0,C 180,E1 -11764.869,E2 -11764.869} C_VEL
LIN {X 0,Y 402.343,Z 352.651,A -85,B 0,C 180,E1 -11765.364,E2 -11765.364} C_VEL
LIN {X 0,Y 401.708,Z 365.636,A -85,B 0,C 180,E1 -11765.962,E2 -11765.962} C_VEL
LIN {X 0,Y 400.785,Z 379.175,A -85,B 0,C 180,E1 -11766.761,E2 -11766.761} C_VEL
LIN {X 0,Y 399.551,Z 392.881,A -85,B 0,C 180,E1 -11767.778,E2 -11767.778} C_VEL
LIN {X 0,Y 398.011,Z 406.674,A -85,B 0,C 180,E1 -11769.048,E2 -11769.048} C_VEL
LIN {X 0,Y 396.56,Z 419.093,A -85,B 0,C 180,E1 -11770.456,E2 -11770.456} C_VEL
LIN {X 0,Y 395.793,Z 426.121,A -85,B 0,C 180,E1 -11771.389,E2 -11771.389} C_VEL
LIN {X 0,Y 394.597,Z 430.367,A -85,B 0,C 180,E1 -11771.963,E2 -11771.963} C_VEL
LIN {X 0,Y 390.949,Z 437.152,A -85,B 0,C 180,E1 -11772.881,E2 -11772.881} C_VEL
LIN {X 0,Y 387.322,Z 443.539,A -85,B 0,C 180,E1 -11773.865,E2 -11773.865} C_VEL
LIN {X 0,Y 386.168,Z 447.071,A -85,B 0,C 180,E1 -11774.534,E2 -11774.534} C_VEL
LIN {X 0,Y 384.992,Z 455.836,A -85,B 0,C 180,E1 -11776.54,E2 -11776.54} C_VEL
LIN {X 0,Y 384.049,Z 462.437,A -85,B 0,C 180,E1 -11778.386,E2 -11778.386} C_VEL
LIN {X 0,Y 383.289,Z 468.533,A -85,B 0,C 180,E1 -11780.5,E2 -11780.5} C_VEL
LIN {X 0,Y 382.729,Z 473.244,A -85,B 0,C 180,E1 -11782.613,E2 -11782.613} C_VEL
LIN {X 0,Y 382.433,Z 476.69,A -85,B 0,C 180,E1 -11784.727,E2 -11784.727} C_VEL
LIN {X 0,Y 382.23,Z 478.964,A -85,B 0,C 180,E1 -11786.837,E2 -11786.837} C_VEL
LIN {X 0,Y 381.981,Z 480.133,A -85,B 0,C 180,E1 -11788.944,E2 -11788.944} C_VEL
LIN {X 0,Y 381.981,Z 480.147,A -85,B 0,C 180,E1 -11791.053,E2 -11791.053} C_VEL
LIN {X 0,Y 382.228,Z 479.034,A -85,B 0,C 180,E1 -11793.161,E2 -11793.161} C_VEL
LIN {X 0,Y 382.421,Z 476.821,A -85,B 0,C 180,E1 -11795.271,E2 -11795.271} C_VEL
LIN {X 0,Y 382.741,Z 473.321,A -85,B 0,C 180,E1 -11797.447,E2 -11797.447} C_VEL
LIN {X 0,Y 383.281,Z 468.8,A -85,B 0,C 180,E1 -11799.497,E2 -11799.497} C_VEL
LIN {X 0,Y 384.02,Z 462.769,A -85,B 0,C 180,E1 -11801.612,E2 -11801.612} C_VEL
LIN {X 0,Y 385.097,Z 455.166,A -85,B 0,C 180,E1 -11803.723,E2 -11803.723} C_VEL
LIN {X 0,Y 386.155,Z 447.419,A -85,B 0,C 180,E1 -11805.495,E2 -11805.495} C_VEL
LIN {X 0,Y 387.412,Z 438.789,A -85,B 0,C 180,E1 -11807.143,E2 -11807.143} C_VEL
LIN {X 0,Y 388.792,Z 428.996,A -85,B 0,C 180,E1 -11808.713,E2 -11808.713} C_VEL
LIN {X 0,Y 390.324,Z 416.433,A -85,B 0,C 180,E1 -11810.401,E2 -11810.401} C_VEL
LIN {X 0,Y 391.984,Z 403.134,A -85,B 0,C 180,E1 -11811.839,E2 -11811.839} C_VEL
LIN {X 0,Y 393.428,Z 389.948,A -85,B 0,C 180,E1 -11813,E2 -11813} C_VEL
LIN {X 0,Y 394.615,Z 376.362,A -85,B 0,C 180,E1 -11813.97,E2 -11813.97} C_VEL
LIN {X 0,Y 395.543,Z 361.036,A -85,B 0,C 180,E1 -11814.823,E2 -11814.823} C_VEL
LIN {X 0,Y 396.308,Z 345.712,A -85,B 0,C 180,E1 -11815.433,E2 -11815.433} C_VEL
LIN {X 0,Y 396.744,Z 330.872,A -85,B 0,C 180,E1 -11815.825,E2 -11815.825} C_VEL
LIN {X 0,Y 399.644,Z 195.222,A -85,B 0,C 180,E1 -11818.322,E2 -11818.322} C_VEL
LIN {X 0,Y 391.384,Z 176.777,A -85,B 0,C 180,E1 -11819.37,E2 -11819.37} C_VEL
LIN {X 0,Y 387.722,Z 169.318,A -85,B 0,C 180,E1 -11819.861,E2 -11819.861} C_VEL
LIN {X 0,Y 383.696,Z 156.723,A -85,B 0,C 180,E1 -11822.083,E2 -11822.083} C_VEL
LIN {X 0,Y 383,Z 154.392,A -85,B 0,C 180,E1 -11822.522,E2 -11822.522} C_VEL
LIN {X 0,Y 383.028,Z 154.398,A -85,B 0,C 180,E1 -11826.163,E2 -11826.163} C_VEL
LIN {X 0,Y 383.003,Z 154.378,A -85,B 0,C 180,E1 -11829.957,E2 -11829.957} C_VEL
LIN {X 0,Y 383.026,Z 154.399,A -85,B 0,C 180,E1 -11832.782,E2 -11832.782} C_VEL
LIN {X 0,Y 382.991,Z 154.404,A -85,B 0,C 180,E1 -11835.788,E2 -11835.788} C_VEL
LIN {X 0,Y 383.008,Z 154.399,A -85,B 0,C 180,E1 -11838.79,E2 -11838.79} C_VEL
LIN {X 0,Y 382.995,Z 154.398,A -85,B 0,C 180,E1 -11842.094,E2 -11842.094} C_VEL
LIN {X 0,Y 383.01,Z 154.391,A -85,B 0,C 180,E1 -11845.331,E2 -11845.331} C_VEL
LIN {X 0,Y 383.029,Z 154.397,A -85,B 0,C 180,E1 -11847.852,E2 -11847.852} C_VEL
LIN {X 0,Y 383.054,Z 154.394,A -85,B 0,C 180,E1 -11851.719,E2 -11851.719} C_VEL
LIN {X 0,Y 383.041,Z 154.384,A -85,B 0,C 180,E1 -11855.039,E2 -11855.039} C_VEL
LIN {X 0,Y 382.982,Z 154.404,A -85,B 0,C 180,E1 -11858.468,E2 -11858.468} C_VEL
LIN {X 0,Y 383.078,Z 154.382,A -85,B 0,C 180,E1 -11861.827,E2 -11861.827} C_VEL
LIN {X 0,Y 383.101,Z 154.384,A -85,B 0,C 180,E1 -11865.118,E2 -11865.118} C_VEL
LIN {X 0,Y 383.087,Z 154.38,A -85,B 0,C 180,E1 -11868.357,E2 -11868.357} C_VEL
LIN {X 0,Y 383.293,Z 154.359,A -85,B 0,C 180,E1 -11871.933,E2 -11871.933} C_VEL
LIN {X 0,Y 383.189,Z 154.366,A -85,B 0,C 180,E1 -11874.738,E2 -11874.738} C_VEL
LIN {X 0,Y 383.377,Z 154.352,A -85,B 0,C 180,E1 -11877.899,E2 -11877.899} C_VEL
LIN {X 0,Y 383.51,Z 154.319,A -85,B 0,C 180,E1 -11880,E2 -11880} C_VEL
LIN {X 0,Y 383.242,Z 154.37,A -85,B 0,C 180,E1 -11883.154,E2 -11883.154} C_VEL
LIN {X 0,Y 383.276,Z 154.35,A -85,B 0,C 180,E1 -11886.316,E2 -11886.316} C_VEL
LIN {X 0,Y 383.249,Z 154.36,A -85,B 0,C 180,E1 -11888.436,E2 -11888.436} C_VEL
LIN {X 0,Y 383.087,Z 154.381,A -85,B 0,C 180,E1 -11891.642,E2 -11891.642} C_VEL
LIN {X 0,Y 383.102,Z 154.384,A -85,B 0,C 180,E1 -11894.882,E2 -11894.882} C_VEL
LIN {X 0,Y 383.052,Z 154.382,A -85,B 0,C 180,E1 -11898.174,E2 -11898.174} C_VEL
LIN {X 0,Y 382.983,Z 154.4,A -85,B 0,C 180,E1 -11901.531,E2 -11901.531} C_VEL
LIN {X 0,Y 383.041,Z 154.385,A -85,B 0,C 180,E1 -11904.961,E2 -11904.961} C_VEL
LIN {X 0,Y 383.019,Z 154.395,A -85,B 0,C 180,E1 -11908.271,E2 -11908.271} C_VEL
LIN {X 0,Y 383,Z 154.405,A -85,B 0,C 180,E1 -11912.15,E2 -11912.15} C_VEL
LIN {X 0,Y 383.008,Z 154.393,A -85,B 0,C 180,E1 -11914.669,E2 -11914.669} C_VEL
LIN {X 0,Y 382.992,Z 154.393,A -85,B 0,C 180,E1 -11917.905,E2 -11917.905} C_VEL
LIN {X 0,Y 382.974,Z 154.375,A -85,B 0,C 180,E1 -11921.349,E2 -11921.349} C_VEL
LIN {X 0,Y 382.999,Z 154.403,A -85,B 0,C 180,E1 -11924.306,E2 -11924.306} C_VEL
LIN {X 0,Y 383.067,Z 154.393,A -85,B 0,C 180,E1 -11927.25,E2 -11927.25} C_VEL
LIN {X 0,Y 383.061,Z 154.488,A -85,B 0,C 180,E1 -11931.115,E2 -11931.115} C_VEL
LIN {X 0,Y 389.343,Z 175.454,A -85,B 0,C 180,E1 -11934.57,E2 -11934.57} C_VEL
LIN {X 0,Y 394.441,Z 193.36,A -85,B 0,C 180,E1 -11937.332,E2 -11937.332} C_VEL
LIN {X 0,Y 391.993,Z 216.29,A -85,B 0,C 180,E1 -11940.195,E2 -11940.195} C_VEL
LIN {X 0,Y 391.585,Z 220.042,A -85,B 0,C 180,E1 -11940.649,E2 -11940.649} C_VEL
LIN {X 0,Y 397.258,Z 266.531,A -85,B 0,C 180,E1 -11942.037,E2 -11942.037} C_VEL
LIN {X 0,Y 397.621,Z 273.355,A -85,B 0,C 180,E1 -11942.2,E2 -11942.2} C_VEL
LIN {X 0,Y 394.921,Z 396.827,A -85,B 0,C 180,E1 -11944.471,E2 -11944.471} C_VEL
LIN {X 0,Y 394.07,Z 412.402,A -85,B 0,C 180,E1 -11944.942,E2 -11944.942} C_VEL
LIN {X 0,Y 392.939,Z 426.705,A -85,B 0,C 180,E1 -11945.57,E2 -11945.57} C_VEL
LIN {X 0,Y 391.672,Z 439.345,A -85,B 0,C 180,E1 -11946.295,E2 -11946.295} C_VEL
LIN {X 0,Y 390.166,Z 453.844,A -85,B 0,C 180,E1 -11947.356,E2 -11947.356} C_VEL
LIN {X 0,Y 388.601,Z 466.669,A -85,B 0,C 180,E1 -11948.518,E2 -11948.518} C_VEL
LIN {X 0,Y 387.013,Z 479.628,A -85,B 0,C 180,E1 -11949.956,E2 -11949.956} C_VEL
LIN {X 0,Y 385.808,Z 489.792,A -85,B 0,C 180,E1 -11951.307,E2 -11951.307} C_VEL
LIN {X 0,Y 384.519,Z 500.531,A -85,B 0,C 180,E1 -11952.998,E2 -11952.998} C_VEL
LIN {X 0,Y 383.363,Z 510.362,A -85,B 0,C 180,E1 -11954.858,E2 -11954.858} C_VEL
LIN {X 0,Y 382.644,Z 518.719,A -85,B 0,C 180,E1 -11956.767,E2 -11956.767} C_VEL
LIN {X 0,Y 382.138,Z 526.243,A -85,B 0,C 180,E1 -11958.867,E2 -11958.867} C_VEL
LIN {X 0,Y 381.854,Z 532.341,A -85,B 0,C 180,E1 -11961.001,E2 -11961.001} C_VEL
LIN {X 0,Y 381.919,Z 535.962,A -85,B 0,C 180,E1 -11962.6,E2 -11962.6} C_VEL
LIN {X 0,Y 381.958,Z 539.636,A -85,B 0,C 180,E1 -11964.723,E2 -11964.723} C_VEL
LIN {X 0,Y 382.074,Z 542.062,A -85,B 0,C 180,E1 -11966.838,E2 -11966.838} C_VEL
LIN {X 0,Y 382.099,Z 543.278,A -85,B 0,C 180,E1 -11968.947,E2 -11968.947} C_VEL
LIN {X 0,Y 382.088,Z 543.276,A -85,B 0,C 180,E1 -11971.055,E2 -11971.055} C_VEL
LIN {X 0,Y 382.075,Z 542.058,A -85,B 0,C 180,E1 -11973.165,E2 -11973.165} C_VEL
LIN {X 0,Y 381.958,Z 539.626,A -85,B 0,C 180,E1 -11975.28,E2 -11975.28} C_VEL
LIN {X 0,Y 382.005,Z 537.581,A -85,B 0,C 180,E1 -11976.55,E2 -11976.55} C_VEL
LIN {X 0,Y 381.908,Z 533.599,A -85,B 0,C 180,E1 -11978.467,E2 -11978.467} C_VEL
LIN {X 0,Y 382.055,Z 527.867,A -85,B 0,C 180,E1 -11980.601,E2 -11980.601} C_VEL
LIN {X 0,Y 382.455,Z 520.595,A -85,B 0,C 180,E1 -11982.74,E2 -11982.74} C_VEL
LIN {X 0,Y 383.172,Z 512.825,A -85,B 0,C 180,E1 -11984.609,E2 -11984.609} C_VEL
LIN {X 0,Y 384.196,Z 503.482,A -85,B 0,C 180,E1 -11986.473,E2 -11986.473} C_VEL
LIN {X 0,Y 385.295,Z 493.988,A -85,B 0,C 180,E1 -11988.066,E2 -11988.066} C_VEL
LIN {X 0,Y 386.574,Z 482.713,A -85,B 0,C 180,E1 -11989.655,E2 -11989.655} C_VEL
LIN {X 0,Y 388.138,Z 470.384,A -85,B 0,C 180,E1 -11991.094,E2 -11991.094} C_VEL
LIN {X 0,Y 389.809,Z 456.844,A -85,B 0,C 180,E1 -11992.389,E2 -11992.389} C_VEL
LIN {X 0,Y 391.26,Z 443.619,A -85,B 0,C 180,E1 -11993.412,E2 -11993.412} C_VEL
LIN {X 0,Y 392.713,Z 428.935,A -85,B 0,C 180,E1 -11994.307,E2 -11994.307} C_VEL
LIN {X 0,Y 393.966,Z 413.76,A -85,B 0,C 180,E1 -11994.998,E2 -11994.998} C_VEL
LIN {X 0,Y 394.908,Z 397.694,A -85,B 0,C 180,E1 -11995.498,E2 -11995.498} C_VEL
LIN {X 0,Y 396.017,Z 354.213,A -85,B 0,C 180,E1 -11996.339,E2 -11996.339} C_VEL
LIN {X 0,Y 400.38,Z 271.01,A -85,B 0,C 180,E1 -11998.507,E2 -11998.507} C_VEL
LIN {X 0,Y 399.442,Z 255.57,A -85,B 0,C 180,E1 -11999.148,E2 -11999.148} C_VEL
LIN {X 0,Y 397.87,Z 241.401,A -85,B 0,C 180,E1 -11999.844,E2 -11999.844} C_VEL
LIN {X 0,Y 396.547,Z 232.375,A -85,B 0,C 180,E1 -12000.357,E2 -12000.357} C_VEL
LIN {X 0,Y 401.125,Z 211.023,A -85,B 0,C 180,E1 -12003.499,E2 -12003.499} C_VEL
LIN {X 0,Y 402.443,Z 205.933,A -85,B 0,C 180,E1 -12004.287,E2 -12004.287} C_VEL
LIN {X 0,Y 401.29,Z 200.046,A -85,B 0,C 180,E1 -12005.715,E2 -12005.715} C_VEL
LIN {X 0,Y 399.4,Z 193.508,A -85,B 0,C 180,E1 -12007.643,E2 -12007.643} C_VEL
LIN {X 0,Y 397.77,Z 188.385,A -85,B 0,C 180,E1 -12009.5,E2 -12009.5} C_VEL
LIN {X 0,Y 396.617,Z 185.098,A -85,B 0,C 180,E1 -12010.969,E2 -12010.969} C_VEL
LIN {X 0,Y 395.127,Z 181.467,A -85,B 0,C 180,E1 -12013.176,E2 -12013.176} C_VEL
LIN {X 0,Y 394.1,Z 179.053,A -85,B 0,C 180,E1 -12015.507,E2 -12015.507} C_VEL
LIN {X 0,Y 393.73,Z 178.135,A -85,B 0,C 180,E1 -12017.29,E2 -12017.29} C_VEL
LIN {X 0,Y 393.536,Z 178.063,A -85,B 0,C 180,E1 -12018.642,E2 -12018.642} C_VEL
LIN {X 0,Y 393.568,Z 179.261,A -85,B 0,C 180,E1 -12021.318,E2 -12021.318} C_VEL
LIN {X 0,Y 394.155,Z 181.111,A -85,B 0,C 180,E1 -12023.359,E2 -12023.359} C_VEL
LIN {X 0,Y 395.177,Z 184.841,A -85,B 0,C 180,E1 -12025.93,E2 -12025.93} C_VEL
LIN {X 0,Y 396.304,Z 189.645,A -85,B 0,C 180,E1 -12028.347,E2 -12028.347} C_VEL
LIN {X 0,Y 397.529,Z 196.098,A -85,B 0,C 180,E1 -12030.91,E2 -12030.91} C_VEL
LIN {X 0,Y 398.208,Z 201.402,A -85,B 0,C 180,E1 -12032.686,E2 -12032.686} C_VEL
LIN {X 0,Y 397.969,Z 204.439,A -85,B 0,C 180,E1 -12033.519,E2 -12033.519} C_VEL
LIN {X 0,Y 396.526,Z 211.25,A -85,B 0,C 180,E1 -12035.098,E2 -12035.098} C_VEL
LIN {X 0,Y 400.242,Z 225.362,A -85,B 0,C 180,E1 -12036.273,E2 -12036.273} C_VEL
LIN {X 0,Y 401.898,Z 233.16,A -85,B 0,C 180,E1 -12036.83,E2 -12036.83} C_VEL
LIN {X 0,Y 395.221,Z 319.374,A -85,B 0,C 180,E1 -12039.677,E2 -12039.677} C_VEL
LIN {X 0,Y 394.44,Z 336.368,A -85,B 0,C 180,E1 -12040.324,E2 -12040.324} C_VEL
LIN {X 0,Y 393.622,Z 350.359,A -85,B 0,C 180,E1 -12041.09,E2 -12041.09} C_VEL
LIN {X 0,Y 392.537,Z 363.626,A -85,B 0,C 180,E1 -12042.022,E2 -12042.022} C_VEL
LIN {X 0,Y 391.386,Z 376.249,A -85,B 0,C 180,E1 -12043.169,E2 -12043.169} C_VEL
LIN {X 0,Y 390.215,Z 387.677,A -85,B 0,C 180,E1 -12044.46,E2 -12044.46} C_VEL
LIN {X 0,Y 389.26,Z 396.137,A -85,B 0,C 180,E1 -12045.626,E2 -12045.626} C_VEL
LIN {X 0,Y 388.051,Z 405.456,A -85,B 0,C 180,E1 -12047.182,E2 -12047.182} C_VEL
LIN {X 0,Y 387.026,Z 412.799,A -85,B 0,C 180,E1 -12048.695,E2 -12048.695} C_VEL
LIN {X 0,Y 386.181,Z 418.145,A -85,B 0,C 180,E1 -12050.044,E2 -12050.044} C_VEL
LIN {X 0,Y 385.371,Z 423.134,A -85,B 0,C 180,E1 -12051.611,E2 -12051.611} C_VEL
LIN {X 0,Y 384.771,Z 426.947,A -85,B 0,C 180,E1 -12053.182,E2 -12053.182} C_VEL
LIN {X 0,Y 384.162,Z 429.711,A -85,B 0,C 180,E1 -12054.752,E2 -12054.752} C_VEL
LIN {X 0,Y 383.96,Z 430.993,A -85,B 0,C 180,E1 -12055.801,E2 -12055.801} C_VEL
LIN {X 0,Y 383.709,Z 431.845,A -85,B 0,C 180,E1 -12056.85,E2 -12056.85} C_VEL
LIN {X 0,Y 383.531,Z 432.244,A -85,B 0,C 180,E1 -12057.9,E2 -12057.9} C_VEL
LIN {X 0,Y 383.309,Z 432.247,A -85,B 0,C 180,E1 -12058.95,E2 -12058.95} C_VEL
LIN {X 0,Y 383.158,Z 431.835,A -85,B 0,C 180,E1 -12060,E2 -12060} C_VEL
LIN {X 0,Y 383.168,Z 430.971,A -85,B 0,C 180,E1 -12061.051,E2 -12061.051} C_VEL
LIN {X 0,Y 383.094,Z 429.678,A -85,B 0,C 180,E1 -12062.103,E2 -12062.103} C_VEL
LIN {X 0,Y 383.089,Z 426.938,A -85,B 0,C 180,E1 -12063.682,E2 -12063.682} C_VEL
LIN {X 0,Y 383.232,Z 423.157,A -85,B 0,C 180,E1 -12065.261,E2 -12065.261} C_VEL
LIN {X 0,Y 383.579,Z 417.137,A -85,B 0,C 180,E1 -12067.154,E2 -12067.154} C_VEL
LIN {X 0,Y 383.877,Z 409.757,A -85,B 0,C 180,E1 -12068.952,E2 -12068.952} C_VEL
LIN {X 0,Y 384.393,Z 401.589,A -85,B 0,C 180,E1 -12070.535,E2 -12070.535} C_VEL
LIN {X 0,Y 384.939,Z 391.562,A -85,B 0,C 180,E1 -12072.12,E2 -12072.12} C_VEL
LIN {X 0,Y 385.534,Z 380.1,A -85,B 0,C 180,E1 -12073.574,E2 -12073.574} C_VEL
LIN {X 0,Y 386.215,Z 368.574,A -85,B 0,C 180,E1 -12074.759,E2 -12074.759} C_VEL
LIN {X 0,Y 386.734,Z 355.689,A -85,B 0,C 180,E1 -12075.819,E2 -12075.819} C_VEL
LIN {X 0,Y 387.233,Z 342.322,A -85,B 0,C 180,E1 -12076.678,E2 -12076.678} C_VEL
LIN {X 0,Y 387.605,Z 328.298,A -85,B 0,C 180,E1 -12077.34,E2 -12077.34} C_VEL
LIN {X 0,Y 388.006,Z 313.936,A -85,B 0,C 180,E1 -12077.798,E2 -12077.798} C_VEL
LIN {X 0,Y 390.222,Z 223.04,A -85,B 0,C 180,E1 -12080.02,E2 -12080.02} C_VEL
LIN {X 0,Y 386.726,Z 201.815,A -85,B 0,C 180,E1 -12080.755,E2 -12080.755} C_VEL
LIN {X 0,Y 388.029,Z 184.61,A -85,B 0,C 180,E1 -12084.049,E2 -12084.049} C_VEL
LIN {X 0,Y 388.319,Z 178.827,A -85,B 0,C 180,E1 -12085.185,E2 -12085.185} C_VEL
LIN {X 0,Y 386.335,Z 168.746,A -85,B 0,C 180,E1 -12087.344,E2 -12087.344} C_VEL
LIN {X 0,Y 383.416,Z 156.146,A -85,B 0,C 180,E1 -12090.135,E2 -12090.135} C_VEL
LIN {X 0,Y 382.997,Z 154.403,A -85,B 0,C 180,E1 -12090.536,E2 -12090.536} C_VEL
LIN {X 0,Y 383.009,Z 154.403,A -85,B 0,C 180,E1 -12093.4,E2 -12093.4} C_VEL
LIN {X 0,Y 383.037,Z 154.396,A -85,B 0,C 180,E1 -12096.164,E2 -12096.164} C_VEL
LIN {X 0,Y 382.993,Z 154.392,A -85,B 0,C 180,E1 -12099.96,E2 -12099.96} C_VEL
LIN {X 0,Y 383.011,Z 154.399,A -85,B 0,C 180,E1 -12102.778,E2 -12102.778} C_VEL
LIN {X 0,Y 383.002,Z 154.401,A -85,B 0,C 180,E1 -12105.789,E2 -12105.789} C_VEL
LIN {X 0,Y 382.994,Z 154.407,A -85,B 0,C 180,E1 -12108.795,E2 -12108.795} C_VEL
LIN {X 0,Y 383.003,Z 154.403,A -85,B 0,C 180,E1 -12112.096,E2 -12112.096} C_VEL
LIN {X 0,Y 383.023,Z 154.4,A -85,B 0,C 180,E1 -12115.331,E2 -12115.331} C_VEL
LIN {X 0,Y 383.017,Z 154.593,A -85,B 0,C 180,E1 -12117.613,E2 -12117.613} C_VEL
LIN {X 0,Y 387.689,Z 169.082,A -85,B 0,C 180,E1 -12120.213,E2 -12120.213} C_VEL
LIN {X 0,Y 388.569,Z 171.117,A -85,B 0,C 180,E1 -12120.378,E2 -12120.378} C_VEL
LIN {X 0,Y 396.637,Z 188.17,A -85,B 0,C 180,E1 -12121.399,E2 -12121.399} C_VEL
LIN {X 0,Y 399.608,Z 195.152,A -85,B 0,C 180,E1 -12121.777,E2 -12121.777} C_VEL
LIN {X 0,Y 397.52,Z 293.687,A -85,B 0,C 180,E1 -12123.591,E2 -12123.591} C_VEL
LIN {X 0,Y 396.542,Z 336.588,A -85,B 0,C 180,E1 -12124.404,E2 -12124.404} C_VEL
LIN {X 0,Y 396.022,Z 351.807,A -85,B 0,C 180,E1 -12124.887,E2 -12124.887} C_VEL
LIN {X 0,Y 395.346,Z 364.601,A -85,B 0,C 180,E1 -12125.459,E2 -12125.459} C_VEL
LIN {X 0,Y 394.461,Z 377.836,A -85,B 0,C 180,E1 -12126.226,E2 -12126.226} C_VEL
LIN {X 0,Y 393.173,Z 391.93,A -85,B 0,C 180,E1 -12127.259,E2 -12127.259} C_VEL
LIN {X 0,Y 391.72,Z 404.756,A -85,B 0,C 180,E1 -12128.419,E2 -12128.419} C_VEL
LIN {X 0,Y 390.264,Z 416.983,A -85,B 0,C 180,E1 -12129.771,E2 -12129.771} C_VEL
LIN {X 0,Y 388.866,Z 428.339,A -85,B 0,C 180,E1 -12131.288,E2 -12131.288} C_VEL
LIN {X 0,Y 387.49,Z 438.217,A -85,B 0,C 180,E1 -12132.857,E2 -12132.857} C_VEL
LIN {X 0,Y 386.168,Z 447.071,A -85,B 0,C 180,E1 -12134.534,E2 -12134.534} C_VEL
LIN {X 0,Y 385.04,Z 450.535,A -85,B 0,C 180,E1 -12135.226,E2 -12135.226} C_VEL
LIN {X 0,Y 381.521,Z 455.946,A -85,B 0,C 180,E1 -12136.353,E2 -12136.353} C_VEL
LIN {X 0,Y 378.055,Z 460.871,A -85,B 0,C 180,E1 -12137.544,E2 -12137.544} C_VEL
LIN {X 0,Y 377.03,Z 463.525,A -85,B 0,C 180,E1 -12138.33,E2 -12138.33} C_VEL
LIN {X 0,Y 376.294,Z 469.119,A -85,B 0,C 180,E1 -12140.322,E2 -12140.322} C_VEL
LIN {X 0,Y 375.721,Z 473.828,A -85,B 0,C 180,E1 -12142.475,E2 -12142.475} C_VEL
LIN {X 0,Y 375.368,Z 477.276,A -85,B 0,C 180,E1 -12144.627,E2 -12144.627} C_VEL
LIN {X 0,Y 375.166,Z 479.549,A -85,B 0,C 180,E1 -12146.777,E2 -12146.777} C_VEL
LIN {X 0,Y 374.933,Z 480.715,A -85,B 0,C 180,E1 -12148.925,E2 -12148.925} C_VEL
LIN {X 0,Y 374.933,Z 480.729,A -85,B 0,C 180,E1 -12151.073,E2 -12151.073} C_VEL
LIN {X 0,Y 375.164,Z 479.618,A -85,B 0,C 180,E1 -12153.22,E2 -12153.22} C_VEL
LIN {X 0,Y 375.355,Z 477.406,A -85,B 0,C 180,E1 -12155.37,E2 -12155.37} C_VEL
LIN {X 0,Y 375.718,Z 474.025,A -85,B 0,C 180,E1 -12157.522,E2 -12157.522} C_VEL
LIN {X 0,Y 376.286,Z 469.384,A -85,B 0,C 180,E1 -12159.676,E2 -12159.676} C_VEL
LIN {X 0,Y 377.074,Z 463.352,A -85,B 0,C 180,E1 -12161.829,E2 -12161.829} C_VEL
LIN {X 0,Y 378.221,Z 455.747,A -85,B 0,C 180,E1 -12163.977,E2 -12163.977} C_VEL
LIN {X 0,Y 379.296,Z 448.162,A -85,B 0,C 180,E1 -12165.748,E2 -12165.748} C_VEL
LIN {X 0,Y 380.652,Z 439.366,A -85,B 0,C 180,E1 -12167.457,E2 -12167.457} C_VEL
LIN {X 0,Y 382.096,Z 429.571,A -85,B 0,C 180,E1 -12169.054,E2 -12169.054} C_VEL
LIN {X 0,Y 383.669,Z 417.259,A -85,B 0,C 180,E1 -12170.737,E2 -12170.737} C_VEL
LIN {X 0,Y 385.247,Z 405.022,A -85,B 0,C 180,E1 -12172.1,E2 -12172.1} C_VEL
LIN {X 0,Y 386.782,Z 392.106,A -85,B 0,C 180,E1 -12173.277,E2 -12173.277} C_VEL
LIN {X 0,Y 388.052,Z 377.918,A -85,B 0,C 180,E1 -12174.33,E2 -12174.33} C_VEL
LIN {X 0,Y 389.033,Z 364.107,A -85,B 0,C 180,E1 -12175.131,E2 -12175.131} C_VEL
LIN {X 0,Y 389.78,Z 349.114,A -85,B 0,C 180,E1 -12175.783,E2 -12175.783} C_VEL
LIN {X 0,Y 390.277,Z 334.333,A -85,B 0,C 180,E1 -12176.214,E2 -12176.214} C_VEL
LIN {X 0,Y 393.388,Z 198.856,A -85,B 0,C 180,E1 -12178.749,E2 -12178.749} C_VEL
LIN {X 0,Y 393.174,Z 196.699,A -85,B 0,C 180,E1 -12178.81,E2 -12178.81} C_VEL
LIN {X 0,Y 385.502,Z 179.59,A -85,B 0,C 180,E1 -12179.813,E2 -12179.813} C_VEL
LIN {X 0,Y 380.692,Z 169.909,A -85,B 0,C 180,E1 -12180.466,E2 -12180.466} C_VEL
LIN {X 0,Y 375.965,Z 155.274,A -85,B 0,C 180,E1 -12183.122,E2 -12183.122} C_VEL
LIN {X 0,Y 375.959,Z 155.277,A -85,B 0,C 180,E1 -12186.503,E2 -12186.503} C_VEL
LIN {X 0,Y 375.982,Z 155.252,A -85,B 0,C 180,E1 -12189.969,E2 -12189.969} C_VEL
LIN {X 0,Y 375.933,Z 155.276,A -85,B 0,C 180,E1 -12193.763,E2 -12193.763} C_VEL
LIN {X 0,Y 375.953,Z 155.273,A -85,B 0,C 180,E1 -12197.703,E2 -12197.703} C_VEL
LIN {X 0,Y 375.961,Z 155.275,A -85,B 0,C 180,E1 -12200.537,E2 -12200.537} C_VEL
LIN {X 0,Y 375.957,Z 155.279,A -85,B 0,C 180,E1 -12203.494,E2 -12203.494} C_VEL
LIN {X 0,Y 375.955,Z 155.271,A -85,B 0,C 180,E1 -12205.888,E2 -12205.888} C_VEL
LIN {X 0,Y 375.961,Z 155.264,A -85,B 0,C 180,E1 -12209.687,E2 -12209.687} C_VEL
LIN {X 0,Y 375.993,Z 155.273,A -85,B 0,C 180,E1 -12212.141,E2 -12212.141} C_VEL
LIN {X 0,Y 375.996,Z 155.265,A -85,B 0,C 180,E1 -12214.538,E2 -12214.538} C_VEL
LIN {X 0,Y 375.948,Z 155.279,A -85,B 0,C 180,E1 -12218.045,E2 -12218.045} C_VEL
LIN {X 0,Y 376.013,Z 155.259,A -85,B 0,C 180,E1 -12221.473,E2 -12221.473} C_VEL
LIN {X 0,Y 376.049,Z 155.266,A -85,B 0,C 180,E1 -12224.832,E2 -12224.832} C_VEL
LIN {X 0,Y 376.04,Z 155.256,A -85,B 0,C 180,E1 -12228.136,E2 -12228.136} C_VEL
LIN {X 0,Y 376.246,Z 155.237,A -85,B 0,C 180,E1 -12231.877,E2 -12231.877} C_VEL
LIN {X 0,Y 376.161,Z 155.239,A -85,B 0,C 180,E1 -12234.64,E2 -12234.64} C_VEL
LIN {X 0,Y 376.343,Z 155.228,A -85,B 0,C 180,E1 -12237.859,E2 -12237.859} C_VEL
LIN {X 0,Y 376.48,Z 155.194,A -85,B 0,C 180,E1 -12240,E2 -12240} C_VEL
LIN {X 0,Y 376.18,Z 155.249,A -85,B 0,C 180,E1 -12243.213,E2 -12243.213} C_VEL
LIN {X 0,Y 376.235,Z 155.225,A -85,B 0,C 180,E1 -12246.435,E2 -12246.435} C_VEL
LIN {X 0,Y 376.194,Z 155.24,A -85,B 0,C 180,E1 -12248.595,E2 -12248.595} C_VEL
LIN {X 0,Y 376.04,Z 155.258,A -85,B 0,C 180,E1 -12251.864,E2 -12251.864} C_VEL
LIN {X 0,Y 376.05,Z 155.262,A -85,B 0,C 180,E1 -12255.168,E2 -12255.168} C_VEL
LIN {X 0,Y 375.998,Z 155.257,A -85,B 0,C 180,E1 -12258.527,E2 -12258.527} C_VEL
LIN {X 0,Y 375.953,Z 155.277,A -85,B 0,C 180,E1 -12261.955,E2 -12261.955} C_VEL
LIN {X 0,Y 375.996,Z 155.265,A -85,B 0,C 180,E1 -12265.462,E2 -12265.462} C_VEL
LIN {X 0,Y 375.95,Z 155.268,A -85,B 0,C 180,E1 -12269.081,E2 -12269.081} C_VEL
LIN {X 0,Y 375.939,Z 155.278,A -85,B 0,C 180,E1 -12272.829,E2 -12272.829} C_VEL
LIN {X 0,Y 375.949,Z 155.276,A -85,B 0,C 180,E1 -12275.416,E2 -12275.416} C_VEL
LIN {X 0,Y 375.966,Z 155.262,A -85,B 0,C 180,E1 -12278.272,E2 -12278.272} C_VEL
LIN {X 0,Y 375.925,Z 155.256,A -85,B 0,C 180,E1 -12281.602,E2 -12281.602} C_VEL
LIN {X 0,Y 375.972,Z 155.277,A -85,B 0,C 180,E1 -12285.262,E2 -12285.262} C_VEL
LIN {X 0,Y 375.982,Z 155.277,A -85,B 0,C 180,E1 -12288.391,E2 -12288.391} C_VEL
LIN {X 0,Y 376.002,Z 155.32,A -85,B 0,C 180,E1 -12290.645,E2 -12290.645} C_VEL
LIN {X 0,Y 382.006,Z 175.533,A -85,B 0,C 180,E1 -12294.046,E2 -12294.046} C_VEL
LIN {X 0,Y 387.201,Z 193.416,A -85,B 0,C 180,E1 -12296.882,E2 -12296.882} C_VEL
LIN {X 0,Y 387.703,Z 195.622,A -85,B 0,C 180,E1 -12297.213,E2 -12297.213} C_VEL
LIN {X 0,Y 385.094,Z 217.975,A -85,B 0,C 180,E1 -12300.04,E2 -12300.04} C_VEL
LIN {X 0,Y 386.513,Z 230.307,A -85,B 0,C 180,E1 -12300.455,E2 -12300.455} C_VEL
LIN {X 0,Y 391.285,Z 270.191,A -85,B 0,C 180,E1 -12301.655,E2 -12301.655} C_VEL
LIN {X 0,Y 388.94,Z 381.612,A -85,B 0,C 180,E1 -12303.725,E2 -12303.725} C_VEL
LIN {X 0,Y 388.379,Z 400.005,A -85,B 0,C 180,E1 -12304.117,E2 -12304.117} C_VEL
LIN {X 0,Y 387.382,Z 415.055,A -85,B 0,C 180,E1 -12304.622,E2 -12304.622} C_VEL
LIN {X 0,Y 386.235,Z 428.613,A -85,B 0,C 180,E1 -12305.261,E2 -12305.261} C_VEL
LIN {X 0,Y 384.929,Z 441.484,A -85,B 0,C 180,E1 -12306.049,E2 -12306.049} C_VEL
LIN {X 0,Y 383.196,Z 456.41,A -85,B 0,C 180,E1 -12307.206,E2 -12307.206} C_VEL
LIN {X 0,Y 381.61,Z 468.689,A -85,B 0,C 180,E1 -12308.389,E2 -12308.389} C_VEL
LIN {X 0,Y 379.981,Z 481.2,A -85,B 0,C 180,E1 -12309.851,E2 -12309.851} C_VEL
LIN {X 0,Y 378.622,Z 492.443,A -85,B 0,C 180,E1 -12311.442,E2 -12311.442} C_VEL
LIN {X 0,Y 377.246,Z 502.956,A -85,B 0,C 180,E1 -12313.218,E2 -12313.218} C_VEL
LIN {X 0,Y 376.152,Z 512.279,A -85,B 0,C 180,E1 -12315.115,E2 -12315.115} C_VEL
LIN {X 0,Y 375.407,Z 520.038,A -85,B 0,C 180,E1 -12317.019,E2 -12317.019} C_VEL
LIN {X 0,Y 374.98,Z 527.307,A -85,B 0,C 180,E1 -12319.199,E2 -12319.199} C_VEL
LIN {X 0,Y 374.775,Z 533.033,A -85,B 0,C 180,E1 -12321.373,E2 -12321.373} C_VEL
LIN {X 0,Y 374.861,Z 537.373,A -85,B 0,C 180,E1 -12323.543,E2 -12323.543} C_VEL
LIN {X 0,Y 374.876,Z 540.41,A -85,B 0,C 180,E1 -12325.701,E2 -12325.701} C_VEL
LIN {X 0,Y 375.039,Z 542.235,A -85,B 0,C 180,E1 -12327.854,E2 -12327.854} C_VEL
LIN {X 0,Y 375.034,Z 542.852,A -85,B 0,C 180,E1 -12330.001,E2 -12330.001} C_VEL
LIN {X 0,Y 375.039,Z 542.233,A -85,B 0,C 180,E1 -12332.149,E2 -12332.149} C_VEL
LIN {X 0,Y 374.874,Z 540.404,A -85,B 0,C 180,E1 -12334.302,E2 -12334.302} C_VEL
LIN {X 0,Y 374.912,Z 537.247,A -85,B 0,C 180,E1 -12336.525,E2 -12336.525} C_VEL
LIN {X 0,Y 374.81,Z 533.006,A -85,B 0,C 180,E1 -12338.629,E2 -12338.629} C_VEL
LIN {X 0,Y 375.005,Z 527.274,A -85,B 0,C 180,E1 -12340.803,E2 -12340.803} C_VEL
LIN {X 0,Y 375.437,Z 520.001,A -85,B 0,C 180,E1 -12342.983,E2 -12342.983} C_VEL
LIN {X 0,Y 376.207,Z 512.231,A -85,B 0,C 180,E1 -12344.885,E2 -12344.885} C_VEL
LIN {X 0,Y 377.287,Z 502.889,A -85,B 0,C 180,E1 -12346.783,E2 -12346.783} C_VEL
LIN {X 0,Y 378.611,Z 492.384,A -85,B 0,C 180,E1 -12348.557,E2 -12348.557} C_VEL
LIN {X 0,Y 379.848,Z 482.127,A -85,B 0,C 180,E1 -12350.018,E2 -12350.018} C_VEL
LIN {X 0,Y 381.288,Z 470.979,A -85,B 0,C 180,E1 -12351.35,E2 -12351.35} C_VEL
LIN {X 0,Y 382.99,Z 457.697,A -85,B 0,C 180,E1 -12352.667,E2 -12352.667} C_VEL
LIN {X 0,Y 384.514,Z 444.726,A -85,B 0,C 180,E1 -12353.711,E2 -12353.711} C_VEL
LIN {X 0,Y 386.077,Z 429.94,A -85,B 0,C 180,E1 -12354.652,E2 -12354.652} C_VEL
LIN {X 0,Y 387.33,Z 415.472,A -85,B 0,C 180,E1 -12355.348,E2 -12355.348} C_VEL
LIN {X 0,Y 388.348,Z 400.639,A -85,B 0,C 180,E1 -12355.852,E2 -12355.852} C_VEL
LIN {X 0,Y 388.917,Z 380.831,A -85,B 0,C 180,E1 -12356.28,E2 -12356.28} C_VEL
LIN {X 0,Y 389.672,Z 362.617,A -85,B 0,C 180,E1 -12356.694,E2 -12356.694} C_VEL
LIN {X 0,Y 393.604,Z 290.503,A -85,B 0,C 180,E1 -12358.607,E2 -12358.607} C_VEL
LIN {X 0,Y 394.764,Z 270.694,A -85,B 0,C 180,E1 -12359.167,E2 -12359.167} C_VEL
LIN {X 0,Y 393.627,Z 252.625,A -85,B 0,C 180,E1 -12359.976,E2 -12359.976} C_VEL
LIN {X 0,Y 391.847,Z 238.062,A -85,B 0,C 180,E1 -12360.774,E2 -12360.774} C_VEL
LIN {X 0,Y 390.962,Z 231.674,A -85,B 0,C 180,E1 -12361.184,E2 -12361.184} C_VEL
LIN {X 0,Y 395.879,Z 211.164,A -85,B 0,C 180,E1 -12364.31,E2 -12364.31} C_VEL
LIN {X 0,Y 396.427,Z 208.409,A -85,B 0,C 180,E1 -12364.78,E2 -12364.78} C_VEL
LIN {X 0,Y 395.138,Z 202.368,A -85,B 0,C 180,E1 -12366.359,E2 -12366.359} C_VEL
LIN {X 0,Y 393.048,Z 195.055,A -85,B 0,C 180,E1 -12368.744,E2 -12368.744} C_VEL
LIN {X 0,Y 391.288,Z 189.762,A -85,B 0,C 180,E1 -12371.03,E2 -12371.03} C_VEL
LIN {X 0,Y 389.863,Z 186.183,A -85,B 0,C 180,E1 -12373.239,E2 -12373.239} C_VEL
LIN {X 0,Y 388.965,Z 184.104,A -85,B 0,C 180,E1 -12375.197,E2 -12375.197} C_VEL
LIN {X 0,Y 388.585,Z 183.191,A -85,B 0,C 180,E1 -12376.586,E2 -12376.586} C_VEL
LIN {X 0,Y 388.316,Z 182.829,A -85,B 0,C 180,E1 -12377.96,E2 -12377.96} C_VEL
LIN {X 0,Y 388.143,Z 183.021,A -85,B 0,C 180,E1 -12379.508,E2 -12379.508} C_VEL
LIN {X 0,Y 388.355,Z 184.452,A -85,B 0,C 180,E1 -12382.027,E2 -12382.027} C_VEL
LIN {X 0,Y 389.042,Z 186.971,A -85,B 0,C 180,E1 -12384.384,E2 -12384.384} C_VEL
LIN {X 0,Y 389.884,Z 190.483,A -85,B 0,C 180,E1 -12386.599,E2 -12386.599} C_VEL
LIN {X 0,Y 390.672,Z 194.46,A -85,B 0,C 180,E1 -12388.554,E2 -12388.554} C_VEL
LIN {X 0,Y 391.725,Z 200.63,A -85,B 0,C 180,E1 -12391.026,E2 -12391.026} C_VEL
LIN {X 0,Y 392.123,Z 204.087,A -85,B 0,C 180,E1 -12392.225,E2 -12392.225} C_VEL
LIN {X 0,Y 392.03,Z 206.998,A -85,B 0,C 180,E1 -12393.086,E2 -12393.086} C_VEL
LIN {X 0,Y 390.92,Z 212.098,A -85,B 0,C 180,E1 -12394.282,E2 -12394.282} C_VEL
LIN {X 0,Y 394.549,Z 225.805,A -85,B 0,C 180,E1 -12395.514,E2 -12395.514} C_VEL
LIN {X 0,Y 396.447,Z 234.741,A -85,B 0,C 180,E1 -12396.199,E2 -12396.199} C_VEL
LIN {X 0,Y 389.29,Z 321.15,A -85,B 0,C 180,E1 -12399.146,E2 -12399.146} C_VEL
LIN {X 0,Y 388.489,Z 336.729,A -85,B 0,C 180,E1 -12399.758,E2 -12399.758} C_VEL
LIN {X 0,Y 387.599,Z 350.899,A -85,B 0,C 180,E1 -12400.542,E2 -12400.542} C_VEL
LIN {X 0,Y 386.449,Z 364.076,A -85,B 0,C 180,E1 -12401.478,E2 -12401.478} C_VEL
LIN {X 0,Y 385.205,Z 376.543,A -85,B 0,C 180,E1 -12402.617,E2 -12402.617} C_VEL
LIN {X 0,Y 383.949,Z 388.094,A -85,B 0,C 180,E1 -12403.927,E2 -12403.927} C_VEL
LIN {X 0,Y 382.866,Z 396.657,A -85,B 0,C 180,E1 -12405.109,E2 -12405.109} C_VEL
LIN {X 0,Y 381.606,Z 406.045,A -85,B 0,C 180,E1 -12406.691,E2 -12406.691} C_VEL
LIN {X 0,Y 380.427,Z 413.685,A -85,B 0,C 180,E1 -12408.275,E2 -12408.275} C_VEL
LIN {X 0,Y 379.384,Z 419.841,A -85,B 0,C 180,E1 -12409.864,E2 -12409.864} C_VEL
LIN {X 0,Y 378.523,Z 424.71,A -85,B 0,C 180,E1 -12411.458,E2 -12411.458} C_VEL
LIN {X 0,Y 377.883,Z 428.401,A -85,B 0,C 180,E1 -12413.057,E2 -12413.057} C_VEL
LIN {X 0,Y 377.244,Z 431.059,A -85,B 0,C 180,E1 -12414.655,E2 -12414.655} C_VEL
LIN {X 0,Y 377.022,Z 432.275,A -85,B 0,C 180,E1 -12415.724,E2 -12415.724} C_VEL
LIN {X 0,Y 376.727,Z 433.043,A -85,B 0,C 180,E1 -12416.792,E2 -12416.792} C_VEL
LIN {X 0,Y 376.554,Z 433.382,A -85,B 0,C 180,E1 -12417.861,E2 -12417.861} C_VEL
LIN {X 0,Y 376.309,Z 433.332,A -85,B 0,C 180,E1 -12418.93,E2 -12418.93} C_VEL
LIN {X 0,Y 376.133,Z 432.86,A -85,B 0,C 180,E1 -12420,E2 -12420} C_VEL
LIN {X 0,Y 376.143,Z 431.908,A -85,B 0,C 180,E1 -12421.071,E2 -12421.071} C_VEL
LIN {X 0,Y 376.07,Z 430.557,A -85,B 0,C 180,E1 -12422.142,E2 -12422.142} C_VEL
LIN {X 0,Y 376.06,Z 427.71,A -85,B 0,C 180,E1 -12423.751,E2 -12423.751} C_VEL
LIN {X 0,Y 376.218,Z 423.816,A -85,B 0,C 180,E1 -12425.36,E2 -12425.36} C_VEL
LIN {X 0,Y 376.537,Z 418.022,A -85,B 0,C 180,E1 -12427.183,E2 -12427.183} C_VEL
LIN {X 0,Y 376.782,Z 411.475,A -85,B 0,C 180,E1 -12428.825,E2 -12428.825} C_VEL
LIN {X 0,Y 377.302,Z 403.295,A -85,B 0,C 180,E1 -12430.464,E2 -12430.464} C_VEL
LIN {X 0,Y 377.873,Z 393.413,A -85,B 0,C 180,E1 -12432.078,E2 -12432.078} C_VEL
LIN {X 0,Y 378.424,Z 383.327,A -85,B 0,C 180,E1 -12433.424,E2 -12433.424} C_VEL
LIN {X 0,Y 379.168,Z 370.876,A -85,B 0,C 180,E1 -12434.765,E2 -12434.765} C_VEL
LIN {X 0,Y 379.697,Z 358.15,A -85,B 0,C 180,E1 -12435.866,E2 -12435.866} C_VEL
LIN {X 0,Y 380.259,Z 344.437,A -85,B 0,C 180,E1 -12436.785,E2 -12436.785} C_VEL
LIN {X 0,Y 380.599,Z 330.248,A -85,B 0,C 180,E1 -12437.496,E2 -12437.496} C_VEL
LIN {X 0,Y 381.031,Z 315.382,A -85,B 0,C 180,E1 -12437.996,E2 -12437.996} C_VEL
LIN {X 0,Y 383.414,Z 223.936,A -85,B 0,C 180,E1 -12440.298,E2 -12440.298} C_VEL
LIN {X 0,Y 379.839,Z 202.129,A -85,B 0,C 180,E1 -12441.06,E2 -12441.06} C_VEL
LIN {X 0,Y 381.264,Z 184.421,A -85,B 0,C 180,E1 -12444.504,E2 -12444.504} C_VEL
LIN {X 0,Y 381.379,Z 179.708,A -85,B 0,C 180,E1 -12445.448,E2 -12445.448} C_VEL
LIN {X 0,Y 378.744,Z 166.925,A -85,B 0,C 180,E1 -12448.241,E2 -12448.241} C_VEL
LIN {X 0,Y 375.957,Z 155.281,A -85,B 0,C 180,E1 -12450.89,E2 -12450.89} C_VEL
LIN {X 0,Y 375.985,Z 155.276,A -85,B 0,C 180,E1 -12454.667,E2 -12454.667} C_VEL
LIN {X 0,Y 375.945,Z 155.279,A -85,B 0,C 180,E1 -12458.263,E2 -12458.263} C_VEL
LIN {X 0,Y 375.928,Z 155.284,A -85,B 0,C 180,E1 -12461.598,E2 -12461.598} C_VEL
LIN {X 0,Y 375.957,Z 155.282,A -85,B 0,C 180,E1 -12465.264,E2 -12465.264} C_VEL
LIN {X 0,Y 375.945,Z 155.28,A -85,B 0,C 180,E1 -12469.132,E2 -12469.132} C_VEL
LIN {X 0,Y 375.968,Z 155.28,A -85,B 0,C 180,E1 -12471.911,E2 -12471.911} C_VEL
LIN {X 0,Y 375.985,Z 155.277,A -85,B 0,C 180,E1 -12475.332,E2 -12475.332} C_VEL
LIN {X 0,Y 375.96,Z 155.413,A -85,B 0,C 180,E1 -12477.012,E2 -12477.012} C_VEL
LIN {X 0,Y 380.652,Z 169.72,A -85,B 0,C 180,E1 -12479.612,E2 -12479.612} C_VEL
LIN {X 0,Y 382.197,Z 172.925,A -85,B 0,C 180,E1 -12479.861,E2 -12479.861} C_VEL
LIN {X 0,Y 390.733,Z 190.859,A -85,B 0,C 180,E1 -12480.972,E2 -12480.972} C_VEL
LIN {X 0,Y 393.431,Z 197.188,A -85,B 0,C 180,E1 -12481.325,E2 -12481.325} C_VEL
LIN {X 0,Y 391.029,Z 299.519,A -85,B 0,C 180,E1 -12483.226,E2 -12483.226} C_VEL
LIN {X 0,Y 390.166,Z 337.11,A -85,B 0,C 180,E1 -12483.955,E2 -12483.955} C_VEL
LIN {X 0,Y 389.633,Z 352.488,A -85,B 0,C 180,E1 -12484.451,E2 -12484.451} C_VEL
LIN {X 0,Y 388.925,Z 365.358,A -85,B 0,C 180,E1 -12485.038,E2 -12485.038} C_VEL
LIN {X 0,Y 388.006,Z 378.404,A -85,B 0,C 180,E1 -12485.806,E2 -12485.806} C_VEL
LIN {X 0,Y 386.663,Z 392.504,A -85,B 0,C 180,E1 -12486.854,E2 -12486.854} C_VEL
LIN {X 0,Y 385.149,Z 405.333,A -85,B 0,C 180,E1 -12488.032,E2 -12488.032} C_VEL
LIN {X 0,Y 383.617,Z 417.683,A -85,B 0,C 180,E1 -12489.421,E2 -12489.421} C_VEL
LIN {X 0,Y 382.177,Z 428.919,A -85,B 0,C 180,E1 -12490.948,E2 -12490.948} C_VEL
LIN {X 0,Y 380.712,Z 438.802,A -85,B 0,C 180,E1 -12492.543,E2 -12492.543} C_VEL
LIN {X 0,Y 379.257,Z 448.288,A -85,B 0,C 180,E1 -12494.379,E2 -12494.379} C_VEL
LIN {X 0,Y 378.097,Z 456.422,A -85,B 0,C 180,E1 -12496.29,E2 -12496.29} C_VEL
LIN {X 0,Y 377.03,Z 463.525,A -85,B 0,C 180,E1 -12498.33,E2 -12498.33} C_VEL
LIN {X 0,Y 376.045,Z 466.045,A -85,B 0,C 180,E1 -12499.13,E2 -12499.13} C_VEL
LIN {X 0,Y 371.337,Z 471.348,A -85,B 0,C 180,E1 -12500.962,E2 -12500.962} C_VEL
LIN {X 0,Y 369.093,Z 473.893,A -85,B 0,C 180,E1 -12502.072,E2 -12502.072} C_VEL
LIN {X 0,Y 368.609,Z 474.983,A -85,B 0,C 180,E1 -12502.657,E2 -12502.657} C_VEL
LIN {X 0,Y 368.305,Z 477.863,A -85,B 0,C 180,E1 -12504.524,E2 -12504.524} C_VEL
LIN {X 0,Y 368.105,Z 480.134,A -85,B 0,C 180,E1 -12506.715,E2 -12506.715} C_VEL
LIN {X 0,Y 367.886,Z 481.298,A -85,B 0,C 180,E1 -12508.904,E2 -12508.904} C_VEL
LIN {X 0,Y 367.885,Z 481.312,A -85,B 0,C 180,E1 -12511.093,E2 -12511.093} C_VEL
LIN {X 0,Y 368.102,Z 480.203,A -85,B 0,C 180,E1 -12513.282,E2 -12513.282} C_VEL
LIN {X 0,Y 368.293,Z 477.992,A -85,B 0,C 180,E1 -12515.474,E2 -12515.474} C_VEL
LIN {X 0,Y 368.711,Z 474.608,A -85,B 0,C 180,E1 -12517.666,E2 -12517.666} C_VEL
LIN {X 0,Y 369.307,Z 469.967,A -85,B 0,C 180,E1 -12519.86,E2 -12519.86} C_VEL
LIN {X 0,Y 370.14,Z 463.934,A -85,B 0,C 180,E1 -12522.054,E2 -12522.054} C_VEL
LIN {X 0,Y 371.355,Z 456.327,A -85,B 0,C 180,E1 -12524.241,E2 -12524.241} C_VEL
LIN {X 0,Y 372.55,Z 448.214,A -85,B 0,C 180,E1 -12526.154,E2 -12526.154} C_VEL
LIN {X 0,Y 374.111,Z 438.402,A -85,B 0,C 180,E1 -12528.056,E2 -12528.056} C_VEL
LIN {X 0,Y 375.67,Z 428.364,A -85,B 0,C 180,E1 -12529.677,E2 -12529.677} C_VEL
LIN {X 0,Y 377.241,Z 416.68,A -85,B 0,C 180,E1 -12531.257,E2 -12531.257} C_VEL
LIN {X 0,Y 378.882,Z 404.267,A -85,B 0,C 180,E1 -12532.636,E2 -12532.636} C_VEL
LIN {X 0,Y 380.454,Z 391.068,A -85,B 0,C 180,E1 -12533.832,E2 -12533.832} C_VEL
LIN {X 0,Y 381.761,Z 377.463,A -85,B 0,C 180,E1 -12534.831,E2 -12534.831} C_VEL
LIN {X 0,Y 382.753,Z 362.101,A -85,B 0,C 180,E1 -12535.712,E2 -12535.712} C_VEL
LIN {X 0,Y 383.548,Z 347.784,A -85,B 0,C 180,E1 -12536.307,E2 -12536.307} C_VEL
LIN {X 0,Y 384.044,Z 331.782,A -85,B 0,C 180,E1 -12536.746,E2 -12536.746} C_VEL
LIN {X 0,Y 387.197,Z 200.511,A -85,B 0,C 180,E1 -12539.227,E2 -12539.227} C_VEL
LIN {X 0,Y 387.005,Z 198.798,A -85,B 0,C 180,E1 -12539.279,E2 -12539.279} C_VEL
LIN {X 0,Y 379.921,Z 182.98,A -85,B 0,C 180,E1 -12540.232,E2 -12540.232} C_VEL
LIN {X 0,Y 373.726,Z 170.616,A -85,B 0,C 180,E1 -12541.076,E2 -12541.076} C_VEL
LIN {X 0,Y 368.925,Z 156.161,A -85,B 0,C 180,E1 -12543.738,E2 -12543.738} C_VEL
LIN {X 0,Y 368.914,Z 156.158,A -85,B 0,C 180,E1 -12547.56,E2 -12547.56} C_VEL
LIN {X 0,Y 368.906,Z 156.132,A -85,B 0,C 180,E1 -12550.368,E2 -12550.368} C_VEL
LIN {X 0,Y 368.889,Z 156.155,A -85,B 0,C 180,E1 -12553.617,E2 -12553.617} C_VEL
LIN {X 0,Y 368.896,Z 156.157,A -85,B 0,C 180,E1 -12556.697,E2 -12556.697} C_VEL
LIN {X 0,Y 368.945,Z 156.152,A -85,B 0,C 180,E1 -12559.634,E2 -12559.634} C_VEL
LIN {X 0,Y 368.895,Z 156.161,A -85,B 0,C 180,E1 -12563.143,E2 -12563.143} C_VEL
LIN {X 0,Y 368.892,Z 156.153,A -85,B 0,C 180,E1 -12566.461,E2 -12566.461} C_VEL
LIN {X 0,Y 368.915,Z 156.14,A -85,B 0,C 180,E1 -12570.31,E2 -12570.31} C_VEL
LIN {X 0,Y 368.972,Z 156.145,A -85,B 0,C 180,E1 -12573.534,E2 -12573.534} C_VEL
LIN {X 0,Y 368.946,Z 156.143,A -85,B 0,C 180,E1 -12576.42,E2 -12576.42} C_VEL
LIN {X 0,Y 368.926,Z 156.145,A -85,B 0,C 180,E1 -12579.946,E2 -12579.946} C_VEL
LIN {X 0,Y 368.966,Z 156.15,A -85,B 0,C 180,E1 -12583.398,E2 -12583.398} C_VEL
LIN {X 0,Y 369.047,Z 156.123,A -85,B 0,C 180,E1 -12586.79,E2 -12586.79} C_VEL
LIN {X 0,Y 369.057,Z 156.137,A -85,B 0,C 180,E1 -12590.131,E2 -12590.131} C_VEL
LIN {X 0,Y 369.177,Z 156.113,A -85,B 0,C 180,E1 -12592.342,E2 -12592.342} C_VEL
LIN {X 0,Y 369.134,Z 156.113,A -85,B 0,C 180,E1 -12594.537,E2 -12594.537} C_VEL
LIN {X 0,Y 369.308,Z 156.104,A -85,B 0,C 180,E1 -12597.819,E2 -12597.819} C_VEL
LIN {X 0,Y 369.449,Z 156.069,A -85,B 0,C 180,E1 -12600,E2 -12600} C_VEL
LIN {X 0,Y 369.308,Z 156.099,A -85,B 0,C 180,E1 -12602.181,E2 -12602.181} C_VEL
LIN {X 0,Y 369.197,Z 156.101,A -85,B 0,C 180,E1 -12606.558,E2 -12606.558} C_VEL
LIN {X 0,Y 369.127,Z 156.123,A -85,B 0,C 180,E1 -12608.761,E2 -12608.761} C_VEL
LIN {X 0,Y 368.995,Z 156.131,A -85,B 0,C 180,E1 -12612.094,E2 -12612.094} C_VEL
LIN {X 0,Y 368.99,Z 156.141,A -85,B 0,C 180,E1 -12615.465,E2 -12615.465} C_VEL
LIN {X 0,Y 368.947,Z 156.133,A -85,B 0,C 180,E1 -12618.895,E2 -12618.895} C_VEL
LIN {X 0,Y 368.922,Z 156.153,A -85,B 0,C 180,E1 -12622.396,E2 -12622.396} C_VEL
LIN {X 0,Y 368.989,Z 156.14,A -85,B 0,C 180,E1 -12625.981,E2 -12625.981} C_VEL
LIN {X 0,Y 368.904,Z 156.144,A -85,B 0,C 180,E1 -12629.691,E2 -12629.691} C_VEL
LIN {X 0,Y 368.887,Z 156.155,A -85,B 0,C 180,E1 -12633.044,E2 -12633.044} C_VEL
LIN {X 0,Y 368.909,Z 156.159,A -85,B 0,C 180,E1 -12636.198,E2 -12636.198} C_VEL
LIN {X 0,Y 368.895,Z 156.132,A -85,B 0,C 180,E1 -12638.954,E2 -12638.954} C_VEL
LIN {X 0,Y 368.872,Z 156.141,A -85,B 0,C 180,E1 -12642.01,E2 -12642.01} C_VEL
LIN {X 0,Y 368.947,Z 156.152,A -85,B 0,C 180,E1 -12645.189,E2 -12645.189} C_VEL
LIN {X 0,Y 368.934,Z 156.155,A -85,B 0,C 180,E1 -12648.187,E2 -12648.187} C_VEL
LIN {X 0,Y 368.97,Z 156.197,A -85,B 0,C 180,E1 -12650.169,E2 -12650.169} C_VEL
LIN {X 0,Y 375.577,Z 178.525,A -85,B 0,C 180,E1 -12654.006,E2 -12654.006} C_VEL
LIN {X 0,Y 380.67,Z 196.325,A -85,B 0,C 180,E1 -12656.863,E2 -12656.863} C_VEL
LIN {X 0,Y 380.859,Z 197.387,A -85,B 0,C 180,E1 -12657.021,E2 -12657.021} C_VEL
LIN {X 0,Y 378.588,Z 215.879,A -85,B 0,C 180,E1 -12659.402,E2 -12659.402} C_VEL
LIN {X 0,Y 379.271,Z 222.89,A -85,B 0,C 180,E1 -12659.686,E2 -12659.686} C_VEL
LIN {X 0,Y 384.519,Z 266.57,A -85,B 0,C 180,E1 -12661.044,E2 -12661.044} C_VEL
LIN {X 0,Y 385.033,Z 273.729,A -85,B 0,C 180,E1 -12661.234,E2 -12661.234} C_VEL
LIN {X 0,Y 382.148,Z 395.863,A -85,B 0,C 180,E1 -12663.553,E2 -12663.553} C_VEL
LIN {X 0,Y 381.255,Z 411.348,A -85,B 0,C 180,E1 -12664.038,E2 -12664.038} C_VEL
LIN {X 0,Y 379.898,Z 426.893,A -85,B 0,C 180,E1 -12664.747,E2 -12664.747} C_VEL
LIN {X 0,Y 378.347,Z 440.916,A -85,B 0,C 180,E1 -12665.605,E2 -12665.605} C_VEL
LIN {X 0,Y 376.802,Z 454.288,A -85,B 0,C 180,E1 -12666.652,E2 -12666.652} C_VEL
LIN {X 0,Y 375.095,Z 466.811,A -85,B 0,C 180,E1 -12667.849,E2 -12667.849} C_VEL
LIN {X 0,Y 373.548,Z 478.464,A -85,B 0,C 180,E1 -12669.201,E2 -12669.201} C_VEL
LIN {X 0,Y 372.09,Z 489.001,A -85,B 0,C 180,E1 -12670.652,E2 -12670.652} C_VEL
LIN {X 0,Y 370.759,Z 499.354,A -85,B 0,C 180,E1 -12672.346,E2 -12672.346} C_VEL
LIN {X 0,Y 369.459,Z 509.181,A -85,B 0,C 180,E1 -12674.274,E2 -12674.274} C_VEL
LIN {X 0,Y 368.638,Z 517.598,A -85,B 0,C 180,E1 -12676.271,E2 -12676.271} C_VEL
LIN {X 0,Y 368.018,Z 525.058,A -85,B 0,C 180,E1 -12678.434,E2 -12678.434} C_VEL
LIN {X 0,Y 367.703,Z 531.16,A -85,B 0,C 180,E1 -12680.652,E2 -12680.652} C_VEL
LIN {X 0,Y 367.757,Z 535.858,A -85,B 0,C 180,E1 -12682.866,E2 -12682.866} C_VEL
LIN {X 0,Y 367.8,Z 538.462,A -85,B 0,C 180,E1 -12684.519,E2 -12684.519} C_VEL
LIN {X 0,Y 367.934,Z 540.892,A -85,B 0,C 180,E1 -12686.716,E2 -12686.716} C_VEL
LIN {X 0,Y 367.986,Z 542.112,A -85,B 0,C 180,E1 -12688.907,E2 -12688.907} C_VEL
LIN {X 0,Y 367.977,Z 542.11,A -85,B 0,C 180,E1 -12691.096,E2 -12691.096} C_VEL
LIN {X 0,Y 367.934,Z 540.887,A -85,B 0,C 180,E1 -12693.286,E2 -12693.286} C_VEL
LIN {X 0,Y 367.808,Z 538.451,A -85,B 0,C 180,E1 -12695.484,E2 -12695.484} C_VEL
LIN {X 0,Y 367.771,Z 535.839,A -85,B 0,C 180,E1 -12697.137,E2 -12697.137} C_VEL
LIN {X 0,Y 367.77,Z 531.133,A -85,B 0,C 180,E1 -12699.349,E2 -12699.349} C_VEL
LIN {X 0,Y 368.047,Z 525.025,A -85,B 0,C 180,E1 -12701.568,E2 -12701.568} C_VEL
LIN {X 0,Y 368.636,Z 517.555,A -85,B 0,C 180,E1 -12703.732,E2 -12703.732} C_VEL
LIN {X 0,Y 369.485,Z 509.124,A -85,B 0,C 180,E1 -12705.728,E2 -12705.728} C_VEL
LIN {X 0,Y 370.775,Z 499.281,A -85,B 0,C 180,E1 -12707.656,E2 -12707.656} C_VEL
LIN {X 0,Y 371.897,Z 490.485,A -85,B 0,C 180,E1 -12709.112,E2 -12709.112} C_VEL
LIN {X 0,Y 373.496,Z 478.341,A -85,B 0,C 180,E1 -12710.805,E2 -12710.805} C_VEL
LIN {X 0,Y 375.307,Z 465.371,A -85,B 0,C 180,E1 -12712.285,E2 -12712.285} C_VEL
LIN {X 0,Y 376.844,Z 454.124,A -85,B 0,C 180,E1 -12713.349,E2 -12713.349} C_VEL
LIN {X 0,Y 378.37,Z 441.063,A -85,B 0,C 180,E1 -12714.37,E2 -12714.37} C_VEL
LIN {X 0,Y 379.91,Z 426.601,A -85,B 0,C 180,E1 -12715.255,E2 -12715.255} C_VEL
LIN {X 0,Y 381.17,Z 411.824,A -85,B 0,C 180,E1 -12715.935,E2 -12715.935} C_VEL
LIN {X 0,Y 382.134,Z 396.658,A -85,B 0,C 180,E1 -12716.415,E2 -12716.415} C_VEL
LIN {X 0,Y 384.428,Z 350.347,A -85,B 0,C 180,E1 -12717.603,E2 -12717.603} C_VEL
LIN {X 0,Y 388.979,Z 277.55,A -85,B 0,C 180,E1 -12719.635,E2 -12719.635} C_VEL
LIN {X 0,Y 389.264,Z 270.896,A -85,B 0,C 180,E1 -12719.848,E2 -12719.848} C_VEL
LIN {X 0,Y 388.241,Z 253.505,A -85,B 0,C 180,E1 -12720.663,E2 -12720.663} C_VEL
LIN {X 0,Y 386.445,Z 238.099,A -85,B 0,C 180,E1 -12721.56,E2 -12721.56} C_VEL
LIN {X 0,Y 385.518,Z 231.203,A -85,B 0,C 180,E1 -12722.032,E2 -12722.032} C_VEL
LIN {X 0,Y 390.247,Z 213.088,A -85,B 0,C 180,E1 -12724.876,E2 -12724.876} C_VEL
LIN {X 0,Y 390.524,Z 211.557,A -85,B 0,C 180,E1 -12725.163,E2 -12725.163} C_VEL
LIN {X 0,Y 389.471,Z 206.443,A -85,B 0,C 180,E1 -12726.548,E2 -12726.548} C_VEL
LIN {X 0,Y 387.633,Z 199.729,A -85,B 0,C 180,E1 -12728.775,E2 -12728.775} C_VEL
LIN {X 0,Y 386.038,Z 194.731,A -85,B 0,C 180,E1 -12730.951,E2 -12730.951} C_VEL
LIN {X 0,Y 384.715,Z 191.25,A -85,B 0,C 180,E1 -12733.053,E2 -12733.053} C_VEL
LIN {X 0,Y 384.018,Z 189.593,A -85,B 0,C 180,E1 -12734.459,E2 -12734.459} C_VEL
LIN {X 0,Y 383.506,Z 188.429,A -85,B 0,C 180,E1 -12735.863,E2 -12735.863} C_VEL
LIN {X 0,Y 383.176,Z 187.742,A -85,B 0,C 180,E1 -12737.263,E2 -12737.263} C_VEL
LIN {X 0,Y 382.884,Z 187.639,A -85,B 0,C 180,E1 -12738.815,E2 -12738.815} C_VEL
LIN {X 0,Y 382.859,Z 188.657,A -85,B 0,C 180,E1 -12741.382,E2 -12741.382} C_VEL
LIN {X 0,Y 383.167,Z 189.685,A -85,B 0,C 180,E1 -12742.751,E2 -12742.751} C_VEL
LIN {X 0,Y 383.501,Z 191.162,A -85,B 0,C 180,E1 -12744.096,E2 -12744.096} C_VEL
LIN {X 0,Y 384.096,Z 193.928,A -85,B 0,C 180,E1 -12746.02,E2 -12746.02} C_VEL
LIN {X 0,Y 384.805,Z 197.693,A -85,B 0,C 180,E1 -12748.018,E2 -12748.018} C_VEL
LIN {X 0,Y 385.706,Z 203.55,A -85,B 0,C 180,E1 -12750.53,E2 -12750.53} C_VEL
LIN {X 0,Y 386.148,Z 208.687,A -85,B 0,C 180,E1 -12752.348,E2 -12752.348} C_VEL
LIN {X 0,Y 385.884,Z 210.698,A -85,B 0,C 180,E1 -12752.915,E2 -12752.915} C_VEL
LIN {X 0,Y 385.427,Z 212.8,A -85,B 0,C 180,E1 -12753.399,E2 -12753.399} C_VEL
LIN {X 0,Y 389.093,Z 226.971,A -85,B 0,C 180,E1 -12754.763,E2 -12754.763} C_VEL
LIN {X 0,Y 391.099,Z 236.845,A -85,B 0,C 180,E1 -12755.561,E2 -12755.561} C_VEL
LIN {X 0,Y 383.529,Z 321.616,A -85,B 0,C 180,E1 -12758.536,E2 -12758.536} C_VEL
LIN {X 0,Y 382.575,Z 338.378,A -85,B 0,C 180,E1 -12759.22,E2 -12759.22} C_VEL
LIN {X 0,Y 381.559,Z 352.764,A -85,B 0,C 180,E1 -12760.048,E2 -12760.048} C_VEL
LIN {X 0,Y 380.253,Z 366.467,A -85,B 0,C 180,E1 -12761.064,E2 -12761.064} C_VEL
LIN {X 0,Y 378.819,Z 379.536,A -85,B 0,C 180,E1 -12762.314,E2 -12762.314} C_VEL
LIN {X 0,Y 377.613,Z 389.653,A -85,B 0,C 180,E1 -12763.511,E2 -12763.511} C_VEL
LIN {X 0,Y 376.358,Z 398.945,A -85,B 0,C 180,E1 -12764.845,E2 -12764.845} C_VEL
LIN {X 0,Y 374.974,Z 408.113,A -85,B 0,C 180,E1 -12766.451,E2 -12766.451} C_VEL
LIN {X 0,Y 373.741,Z 415.577,A -85,B 0,C 180,E1 -12768.062,E2 -12768.062} C_VEL
LIN {X 0,Y 372.612,Z 421.571,A -85,B 0,C 180,E1 -12769.678,E2 -12769.678} C_VEL
LIN {X 0,Y 371.707,Z 426.3,A -85,B 0,C 180,E1 -12771.3,E2 -12771.3} C_VEL
LIN {X 0,Y 371.002,Z 429.874,A -85,B 0,C 180,E1 -12772.927,E2 -12772.927} C_VEL
LIN {X 0,Y 370.32,Z 432.429,A -85,B 0,C 180,E1 -12774.555,E2 -12774.555} C_VEL
LIN {X 0,Y 370.079,Z 433.545,A -85,B 0,C 180,E1 -12775.644,E2 -12775.644} C_VEL
LIN {X 0,Y 369.767,Z 434.245,A -85,B 0,C 180,E1 -12776.731,E2 -12776.731} C_VEL
LIN {X 0,Y 369.573,Z 434.529,A -85,B 0,C 180,E1 -12777.82,E2 -12777.82} C_VEL
LIN {X 0,Y 369.306,Z 434.421,A -85,B 0,C 180,E1 -12778.91,E2 -12778.91} C_VEL
LIN {X 0,Y 369.107,Z 433.859,A -85,B 0,C 180,E1 -12780,E2 -12780} C_VEL
LIN {X 0,Y 369.117,Z 432.837,A -85,B 0,C 180,E1 -12781.091,E2 -12781.091} C_VEL
LIN {X 0,Y 369.047,Z 431.424,A -85,B 0,C 180,E1 -12782.183,E2 -12782.183} C_VEL
LIN {X 0,Y 369.03,Z 428.466,A -85,B 0,C 180,E1 -12783.822,E2 -12783.822} C_VEL
LIN {X 0,Y 369.204,Z 424.452,A -85,B 0,C 180,E1 -12785.462,E2 -12785.462} C_VEL
LIN {X 0,Y 369.501,Z 418.934,A -85,B 0,C 180,E1 -12787.204,E2 -12787.204} C_VEL
LIN {X 0,Y 369.775,Z 411.683,A -85,B 0,C 180,E1 -12789.021,E2 -12789.021} C_VEL
LIN {X 0,Y 370.312,Z 403.459,A -85,B 0,C 180,E1 -12790.664,E2 -12790.664} C_VEL
LIN {X 0,Y 370.895,Z 393.38,A -85,B 0,C 180,E1 -12792.309,E2 -12792.309} C_VEL
LIN {X 0,Y 371.516,Z 381.868,A -85,B 0,C 180,E1 -12793.818,E2 -12793.818} C_VEL
LIN {X 0,Y 372.257,Z 370.331,A -85,B 0,C 180,E1 -12795.046,E2 -12795.046} C_VEL
LIN {X 0,Y 372.816,Z 356.688,A -85,B 0,C 180,E1 -12796.204,E2 -12796.204} C_VEL
LIN {X 0,Y 373.363,Z 342.981,A -85,B 0,C 180,E1 -12797.105,E2 -12797.105} C_VEL
LIN {X 0,Y 373.77,Z 328.782,A -85,B 0,C 180,E1 -12797.791,E2 -12797.791} C_VEL
LIN {X 0,Y 374.201,Z 314.222,A -85,B 0,C 180,E1 -12798.265,E2 -12798.265} C_VEL
LIN {X 0,Y 376.562,Z 224.677,A -85,B 0,C 180,E1 -12800.583,E2 -12800.583} C_VEL
LIN {X 0,Y 372.98,Z 202.418,A -85,B 0,C 180,E1 -12801.376,E2 -12801.376} C_VEL
LIN {X 0,Y 374.367,Z 185.581,A -85,B 0,C 180,E1 -12804.69,E2 -12804.69} C_VEL
LIN {X 0,Y 374.495,Z 181.248,A -85,B 0,C 180,E1 -12805.571,E2 -12805.571} C_VEL
LIN {X 0,Y 371.753,Z 168.07,A -85,B 0,C 180,E1 -12808.495,E2 -12808.495} C_VEL
LIN {X 0,Y 368.936,Z 156.156,A -85,B 0,C 180,E1 -12811.271,E2 -12811.271} C_VEL
LIN {X 0,Y 368.934,Z 156.155,A -85,B 0,C 180,E1 -12815.001,E2 -12815.001} C_VEL
LIN {X 0,Y 368.886,Z 156.16,A -85,B 0,C 180,E1 -12818.634,E2 -12818.634} C_VEL
LIN {X 0,Y 368.879,Z 156.16,A -85,B 0,C 180,E1 -12822.008,E2 -12822.008} C_VEL
LIN {X 0,Y 368.93,Z 156.155,A -85,B 0,C 180,E1 -12825.182,E2 -12825.182} C_VEL
LIN {X 0,Y 368.888,Z 156.16,A -85,B 0,C 180,E1 -12828.177,E2 -12828.177} C_VEL
LIN {X 0,Y 368.913,Z 156.161,A -85,B 0,C 180,E1 -12831.359,E2 -12831.359} C_VEL
LIN {X 0,Y 368.941,Z 156.153,A -85,B 0,C 180,E1 -12835.146,E2 -12835.146} C_VEL
LIN {X 0,Y 368.95,Z 156.187,A -85,B 0,C 180,E1 -12836.384,E2 -12836.384} C_VEL
LIN {X 0,Y 373.742,Z 170.73,A -85,B 0,C 180,E1 -12839.042,E2 -12839.042} C_VEL
LIN {X 0,Y 382.863,Z 189.265,A -85,B 0,C 180,E1 -12840.269,E2 -12840.269} C_VEL
LIN {X 0,Y 387.153,Z 199.041,A -85,B 0,C 180,E1 -12840.843,E2 -12840.843} C_VEL
LIN {X 0,Y 384.799,Z 298.234,A -85,B 0,C 180,E1 -12842.72,E2 -12842.72} C_VEL
LIN {X 0,Y 383.837,Z 337.628,A -85,B 0,C 180,E1 -12843.492,E2 -12843.492} C_VEL
LIN {X 0,Y 383.303,Z 352.582,A -85,B 0,C 180,E1 -12843.979,E2 -12843.979} C_VEL
LIN {X 0,Y 382.513,Z 366.083,A -85,B 0,C 180,E1 -12844.6,E2 -12844.6} C_VEL
LIN {X 0,Y 381.544,Z 378.974,A -85,B 0,C 180,E1 -12845.369,E2 -12845.369} C_VEL
LIN {X 0,Y 380.166,Z 393.077,A -85,B 0,C 180,E1 -12846.435,E2 -12846.435} C_VEL
LIN {X 0,Y 378.591,Z 405.911,A -85,B 0,C 180,E1 -12847.631,E2 -12847.631} C_VEL
LIN {X 0,Y 376.969,Z 418.399,A -85,B 0,C 180,E1 -12849.06,E2 -12849.06} C_VEL
LIN {X 0,Y 375.5,Z 429.5,A -85,B 0,C 180,E1 -12850.595,E2 -12850.595} C_VEL
LIN {X 0,Y 373.963,Z 439.385,A -85,B 0,C 180,E1 -12852.217,E2 -12852.217} C_VEL
LIN {X 0,Y 372.413,Z 449.005,A -85,B 0,C 180,E1 -12854.113,E2 -12854.113} C_VEL
LIN {X 0,Y 371.203,Z 457.008,A -85,B 0,C 180,E1 -12856.03,E2 -12856.03} C_VEL
LIN {X 0,Y 370.049,Z 464.366,A -85,B 0,C 180,E1 -12858.191,E2 -12858.191} C_VEL
LIN {X 0,Y 369.316,Z 469.704,A -85,B 0,C 180,E1 -12860.137,E2 -12860.137} C_VEL
LIN {X 0,Y 368.69,Z 474.556,A -85,B 0,C 180,E1 -12862.407,E2 -12862.407} C_VEL
LIN {X 0,Y 368.609,Z 474.983,A -85,B 0,C 180,E1 -12862.657,E2 -12862.657} C_VEL
LIN {X 0,Y 367.728,Z 476.556,A -85,B 0,C 180,E1 -12863.537,E2 -12863.537} C_VEL
LIN {X 0,Y 364.667,Z 478.793,A -85,B 0,C 180,E1 -12864.972,E2 -12864.972} C_VEL
LIN {X 0,Y 362.161,Z 480.213,A -85,B 0,C 180,E1 -12866.144,E2 -12866.144} C_VEL
LIN {X 0,Y 361.058,Z 480.994,A -85,B 0,C 180,E1 -12867.059,E2 -12867.059} C_VEL
LIN {X 0,Y 360.948,Z 481.182,A -85,B 0,C 180,E1 -12867.37,E2 -12867.37} C_VEL
LIN {X 0,Y 360.84,Z 481.881,A -85,B 0,C 180,E1 -12868.883,E2 -12868.883} C_VEL
LIN {X 0,Y 360.839,Z 481.894,A -85,B 0,C 180,E1 -12871.115,E2 -12871.115} C_VEL
LIN {X 0,Y 361.044,Z 480.786,A -85,B 0,C 180,E1 -12873.346,E2 -12873.346} C_VEL
LIN {X 0,Y 361.233,Z 478.577,A -85,B 0,C 180,E1 -12875.581,E2 -12875.581} C_VEL
LIN {X 0,Y 361.694,Z 475.192,A -85,B 0,C 180,E1 -12877.816,E2 -12877.816} C_VEL
LIN {X 0,Y 362.335,Z 470.549,A -85,B 0,C 180,E1 -12880.052,E2 -12880.052} C_VEL
LIN {X 0,Y 363.217,Z 464.516,A -85,B 0,C 180,E1 -12882.287,E2 -12882.287} C_VEL
LIN {X 0,Y 364.499,Z 456.907,A -85,B 0,C 180,E1 -12884.515,E2 -12884.515} C_VEL
LIN {X 0,Y 365.743,Z 448.794,A -85,B 0,C 180,E1 -12886.463,E2 -12886.463} C_VEL
LIN {X 0,Y 367.373,Z 438.98,A -85,B 0,C 180,E1 -12888.398,E2 -12888.398} C_VEL
LIN {X 0,Y 369.003,Z 428.94,A -85,B 0,C 180,E1 -12890.047,E2 -12890.047} C_VEL
LIN {X 0,Y 370.61,Z 417.494,A -85,B 0,C 180,E1 -12891.625,E2 -12891.625} C_VEL
LIN {X 0,Y 372.352,Z 404.835,A -85,B 0,C 180,E1 -12893.055,E2 -12893.055} C_VEL
LIN {X 0,Y 374.009,Z 391.627,A -85,B 0,C 180,E1 -12894.269,E2 -12894.269} C_VEL
LIN {X 0,Y 375.362,Z 378.015,A -85,B 0,C 180,E1 -12895.283,E2 -12895.283} C_VEL
LIN {X 0,Y 376.383,Z 362.713,A -85,B 0,C 180,E1 -12896.176,E2 -12896.176} C_VEL
LIN {X 0,Y 377.217,Z 348.294,A -85,B 0,C 180,E1 -12896.783,E2 -12896.783} C_VEL
LIN {X 0,Y 377.743,Z 332.237,A -85,B 0,C 180,E1 -12897.229,E2 -12897.229} C_VEL
LIN {X 0,Y 381.031,Z 202.323,A -85,B 0,C 180,E1 -12899.718,E2 -12899.718} C_VEL
LIN {X 0,Y 380.64,Z 200.237,A -85,B 0,C 180,E1 -12899.797,E2 -12899.797} C_VEL
LIN {X 0,Y 374.001,Z 185.765,A -85,B 0,C 180,E1 -12900.71,E2 -12900.71} C_VEL
LIN {X 0,Y 366.67,Z 171.191,A -85,B 0,C 180,E1 -12901.742,E2 -12901.742} C_VEL
LIN {X 0,Y 361.872,Z 157.034,A -85,B 0,C 180,E1 -12904.403,E2 -12904.403} C_VEL
LIN {X 0,Y 361.865,Z 157.033,A -85,B 0,C 180,E1 -12907.223,E2 -12907.223} C_VEL
LIN {X 0,Y 361.832,Z 157.015,A -85,B 0,C 180,E1 -12910.754,E2 -12910.754} C_VEL
LIN {X 0,Y 361.816,Z 157.032,A -85,B 0,C 180,E1 -12914.366,E2 -12914.366} C_VEL
LIN {X 0,Y 361.849,Z 157.029,A -85,B 0,C 180,E1 -12917.563,E2 -12917.563} C_VEL
LIN {X 0,Y 361.867,Z 157.026,A -85,B 0,C 180,E1 -12920.971,E2 -12920.971} C_VEL
LIN {X 0,Y 361.866,Z 157.028,A -85,B 0,C 180,E1 -12924.654,E2 -12924.654} C_VEL
LIN {X 0,Y 361.851,Z 157.035,A -85,B 0,C 180,E1 -12928.372,E2 -12928.372} C_VEL
LIN {X 0,Y 361.913,Z 157.027,A -85,B 0,C 180,E1 -12932.221,E2 -12932.221} C_VEL
LIN {X 0,Y 361.917,Z 157.016,A -85,B 0,C 180,E1 -12934.709,E2 -12934.709} C_VEL
LIN {X 0,Y 361.879,Z 157.032,A -85,B 0,C 180,E1 -12938.346,E2 -12938.346} C_VEL
LIN {X 0,Y 361.957,Z 157.013,A -85,B 0,C 180,E1 -12942.061,E2 -12942.061} C_VEL
LIN {X 0,Y 361.987,Z 157.008,A -85,B 0,C 180,E1 -12946.101,E2 -12946.101} C_VEL
LIN {X 0,Y 362.021,Z 157.013,A -85,B 0,C 180,E1 -12949.938,E2 -12949.938} C_VEL
LIN {X 0,Y 362.14,Z 156.991,A -85,B 0,C 180,E1 -12952.192,E2 -12952.192} C_VEL
LIN {X 0,Y 362.108,Z 156.987,A -85,B 0,C 180,E1 -12954.431,E2 -12954.431} C_VEL
LIN {X 0,Y 362.272,Z 156.981,A -85,B 0,C 180,E1 -12957.776,E2 -12957.776} C_VEL
LIN {X 0,Y 362.419,Z 156.945,A -85,B 0,C 180,E1 -12960,E2 -12960} C_VEL
LIN {X 0,Y 362.272,Z 156.976,A -85,B 0,C 180,E1 -12962.223,E2 -12962.223} C_VEL
LIN {X 0,Y 362.161,Z 156.976,A -85,B 0,C 180,E1 -12966.686,E2 -12966.686} C_VEL
LIN {X 0,Y 362.063,Z 157.005,A -85,B 0,C 180,E1 -12968.933,E2 -12968.933} C_VEL
LIN {X 0,Y 361.949,Z 157.005,A -85,B 0,C 180,E1 -12972.333,E2 -12972.333} C_VEL
LIN {X 0,Y 361.952,Z 157.012,A -85,B 0,C 180,E1 -12974.621,E2 -12974.621} C_VEL
LIN {X 0,Y 361.945,Z 157.01,A -85,B 0,C 180,E1 -12978.1,E2 -12978.1} C_VEL
LIN {X 0,Y 361.881,Z 157.029,A -85,B 0,C 180,E1 -12981.653,E2 -12981.653} C_VEL
LIN {X 0,Y 361.918,Z 157.017,A -85,B 0,C 180,E1 -12985.291,E2 -12985.291} C_VEL
LIN {X 0,Y 361.898,Z 157.03,A -85,B 0,C 180,E1 -12987.78,E2 -12987.78} C_VEL
LIN {X 0,Y 361.827,Z 157.038,A -85,B 0,C 180,E1 -12991.63,E2 -12991.63} C_VEL
LIN {X 0,Y 361.865,Z 157.03,A -85,B 0,C 180,E1 -12995.346,E2 -12995.346} C_VEL
LIN {X 0,Y 361.861,Z 157.005,A -85,B 0,C 180,E1 -12999.028,E2 -12999.028} C_VEL
LIN {X 0,Y 361.829,Z 157.032,A -85,B 0,C 180,E1 -13002.83,E2 -13002.83} C_VEL
LIN {X 0,Y 361.905,Z 157.031,A -85,B 0,C 180,E1 -13005.932,E2 -13005.932} C_VEL
LIN {X 0,Y 361.925,Z 157.064,A -85,B 0,C 180,E1 -13009.691,E2 -13009.691} C_VEL
LIN {X 0,Y 368.401,Z 179.122,A -85,B 0,C 180,E1 -13013.562,E2 -13013.562} C_VEL
LIN {X 0,Y 373.502,Z 196.798,A -85,B 0,C 180,E1 -13016.466,E2 -13016.466} C_VEL
LIN {X 0,Y 373.983,Z 198.581,A -85,B 0,C 180,E1 -13016.747,E2 -13016.747} C_VEL
LIN {X 0,Y 372.171,Z 213.628,A -85,B 0,C 180,E1 -13018.736,E2 -13018.736} C_VEL
LIN {X 0,Y 372.816,Z 221.214,A -85,B 0,C 180,E1 -13019.078,E2 -13019.078} C_VEL
LIN {X 0,Y 378.615,Z 270.417,A -85,B 0,C 180,E1 -13020.639,E2 -13020.639} C_VEL
LIN {X 0,Y 378.665,Z 279.262,A -85,B 0,C 180,E1 -13020.83,E2 -13020.83} C_VEL
LIN {X 0,Y 375.825,Z 393.912,A -85,B 0,C 180,E1 -13023.035,E2 -13023.035} C_VEL
LIN {X 0,Y 374.963,Z 409.009,A -85,B 0,C 180,E1 -13023.494,E2 -13023.494} C_VEL
LIN {X 0,Y 373.663,Z 423.763,A -85,B 0,C 180,E1 -13024.145,E2 -13024.145} C_VEL
LIN {X 0,Y 372.118,Z 438.053,A -85,B 0,C 180,E1 -13024.996,E2 -13024.996} C_VEL
LIN {X 0,Y 370.457,Z 452.134,A -85,B 0,C 180,E1 -13026.079,E2 -13026.079} C_VEL
LIN {X 0,Y 368.611,Z 464.933,A -85,B 0,C 180,E1 -13027.29,E2 -13027.29} C_VEL
LIN {X 0,Y 366.839,Z 477.882,A -85,B 0,C 180,E1 -13028.803,E2 -13028.803} C_VEL
LIN {X 0,Y 365.211,Z 488.938,A -85,B 0,C 180,E1 -13030.357,E2 -13030.357} C_VEL
LIN {X 0,Y 363.89,Z 498.765,A -85,B 0,C 180,E1 -13032.002,E2 -13032.002} C_VEL
LIN {X 0,Y 362.517,Z 508.589,A -85,B 0,C 180,E1 -13033.965,E2 -13033.965} C_VEL
LIN {X 0,Y 361.617,Z 517.004,A -85,B 0,C 180,E1 -13035.999,E2 -13035.999} C_VEL
LIN {X 0,Y 360.973,Z 524.466,A -85,B 0,C 180,E1 -13038.205,E2 -13038.205} C_VEL
LIN {X 0,Y 360.613,Z 530.568,A -85,B 0,C 180,E1 -13040.466,E2 -13040.466} C_VEL
LIN {X 0,Y 360.67,Z 535.269,A -85,B 0,C 180,E1 -13042.725,E2 -13042.725} C_VEL
LIN {X 0,Y 360.715,Z 537.875,A -85,B 0,C 180,E1 -13044.411,E2 -13044.411} C_VEL
LIN {X 0,Y 360.847,Z 540.305,A -85,B 0,C 180,E1 -13046.652,E2 -13046.652} C_VEL
LIN {X 0,Y 360.932,Z 541.528,A -85,B 0,C 180,E1 -13048.886,E2 -13048.886} C_VEL
LIN {X 0,Y 360.923,Z 541.527,A -85,B 0,C 180,E1 -13051.117,E2 -13051.117} C_VEL
LIN {X 0,Y 360.847,Z 540.3,A -85,B 0,C 180,E1 -13053.351,E2 -13053.351} C_VEL
LIN {X 0,Y 360.729,Z 537.863,A -85,B 0,C 180,E1 -13055.592,E2 -13055.592} C_VEL
LIN {X 0,Y 360.682,Z 535.248,A -85,B 0,C 180,E1 -13057.278,E2 -13057.278} C_VEL
LIN {X 0,Y 360.69,Z 530.54,A -85,B 0,C 180,E1 -13059.535,E2 -13059.535} C_VEL
LIN {X 0,Y 361.004,Z 524.431,A -85,B 0,C 180,E1 -13061.796,E2 -13061.796} C_VEL
LIN {X 0,Y 361.62,Z 516.959,A -85,B 0,C 180,E1 -13064.004,E2 -13064.004} C_VEL
LIN {X 0,Y 362.544,Z 508.529,A -85,B 0,C 180,E1 -13066.037,E2 -13066.037} C_VEL
LIN {X 0,Y 363.902,Z 498.687,A -85,B 0,C 180,E1 -13068.001,E2 -13068.001} C_VEL
LIN {X 0,Y 365.23,Z 488.534,A -85,B 0,C 180,E1 -13069.694,E2 -13069.694} C_VEL
LIN {X 0,Y 366.91,Z 476.673,A -85,B 0,C 180,E1 -13071.343,E2 -13071.343} C_VEL
LIN {X 0,Y 368.657,Z 464.785,A -85,B 0,C 180,E1 -13072.71,E2 -13072.71} C_VEL
LIN {X 0,Y 370.466,Z 451.959,A -85,B 0,C 180,E1 -13073.924,E2 -13073.924} C_VEL
LIN {X 0,Y 372.16,Z 438.139,A -85,B 0,C 180,E1 -13074.981,E2 -13074.981} C_VEL
LIN {X 0,Y 373.689,Z 423.45,A -85,B 0,C 180,E1 -13075.856,E2 -13075.856} C_VEL
LIN {X 0,Y 375.08,Z 407.667,A -85,B 0,C 180,E1 -13076.538,E2 -13076.538} C_VEL
LIN {X 0,Y 376.988,Z 380.011,A -85,B 0,C 180,E1 -13077.441,E2 -13077.441} C_VEL
LIN {X 0,Y 380.655,Z 319.627,A -85,B 0,C 180,E1 -13079.104,E2 -13079.104} C_VEL
LIN {X 0,Y 383.959,Z 273.042,A -85,B 0,C 180,E1 -13080.475,E2 -13080.475} C_VEL
LIN {X 0,Y 383.104,Z 255.46,A -85,B 0,C 180,E1 -13081.33,E2 -13081.33} C_VEL
LIN {X 0,Y 381.421,Z 239.52,A -85,B 0,C 180,E1 -13082.301,E2 -13082.301} C_VEL
LIN {X 0,Y 380.285,Z 230.527,A -85,B 0,C 180,E1 -13082.96,E2 -13082.96} C_VEL
LIN {X 0,Y 384.614,Z 215.162,A -85,B 0,C 180,E1 -13085.463,E2 -13085.463} C_VEL
LIN {X 0,Y 383.784,Z 210.321,A -85,B 0,C 180,E1 -13086.801,E2 -13086.801} C_VEL
LIN {X 0,Y 382.301,Z 204.754,A -85,B 0,C 180,E1 -13088.686,E2 -13088.686} C_VEL
LIN {X 0,Y 380.815,Z 199.782,A -85,B 0,C 180,E1 -13090.829,E2 -13090.829} C_VEL
LIN {X 0,Y 379.909,Z 197.2,A -85,B 0,C 180,E1 -13092.272,E2 -13092.272} C_VEL
LIN {X 0,Y 379.115,Z 195.232,A -85,B 0,C 180,E1 -13093.699,E2 -13093.699} C_VEL
LIN {X 0,Y 378.491,Z 193.794,A -85,B 0,C 180,E1 -13095.122,E2 -13095.122} C_VEL
LIN {X 0,Y 378.064,Z 192.835,A -85,B 0,C 180,E1 -13096.543,E2 -13096.543} C_VEL
LIN {X 0,Y 377.723,Z 192.409,A -85,B 0,C 180,E1 -13098.096,E2 -13098.096} C_VEL
LIN {X 0,Y 377.499,Z 192.972,A -85,B 0,C 180,E1 -13100.729,E2 -13100.729} C_VEL
LIN {X 0,Y 377.837,Z 194.681,A -85,B 0,C 180,E1 -13103.115,E2 -13103.115} C_VEL
LIN {X 0,Y 378.2,Z 196.734,A -85,B 0,C 180,E1 -13104.851,E2 -13104.851} C_VEL
LIN {X 0,Y 378.75,Z 199.462,A -85,B 0,C 180,E1 -13106.618,E2 -13106.618} C_VEL
LIN {X 0,Y 379.408,Z 203.672,A -85,B 0,C 180,E1 -13108.758,E2 -13108.758} C_VEL
LIN {X 0,Y 380.141,Z 209.778,A -85,B 0,C 180,E1 -13111.27,E2 -13111.27} C_VEL
LIN {X 0,Y 380.08,Z 213.435,A -85,B 0,C 180,E1 -13112.448,E2 -13112.448} C_VEL
LIN {X 0,Y 383.698,Z 227.588,A -85,B 0,C 180,E1 -13113.922,E2 -13113.922} C_VEL
LIN {X 0,Y 385.876,Z 238.775,A -85,B 0,C 180,E1 -13114.881,E2 -13114.881} C_VEL
LIN {X 0,Y 377.854,Z 322.559,A -85,B 0,C 180,E1 -13117.91,E2 -13117.91} C_VEL
LIN {X 0,Y 376.768,Z 339.949,A -85,B 0,C 180,E1 -13118.648,E2 -13118.648} C_VEL
LIN {X 0,Y 375.653,Z 354.397,A -85,B 0,C 180,E1 -13119.511,E2 -13119.511} C_VEL
LIN {X 0,Y 374.253,Z 367.762,A -85,B 0,C 180,E1 -13120.53,E2 -13120.53} C_VEL
LIN {X 0,Y 372.633,Z 381.386,A -85,B 0,C 180,E1 -13121.869,E2 -13121.869} C_VEL
LIN {X 0,Y 371.154,Z 392.299,A -85,B 0,C 180,E1 -13123.216,E2 -13123.216} C_VEL
LIN {X 0,Y 369.858,Z 401.309,A -85,B 0,C 180,E1 -13124.572,E2 -13124.572} C_VEL
LIN {X 0,Y 368.369,Z 410.255,A -85,B 0,C 180,E1 -13126.203,E2 -13126.203} C_VEL
LIN {X 0,Y 367.061,Z 417.491,A -85,B 0,C 180,E1 -13127.842,E2 -13127.842} C_VEL
LIN {X 0,Y 365.853,Z 423.311,A -85,B 0,C 180,E1 -13129.485,E2 -13129.485} C_VEL
LIN {X 0,Y 364.883,Z 427.894,A -85,B 0,C 180,E1 -13131.136,E2 -13131.136} C_VEL
LIN {X 0,Y 364.254,Z 430.321,A -85,B 0,C 180,E1 -13132.238,E2 -13132.238} C_VEL
LIN {X 0,Y 363.771,Z 432.293,A -85,B 0,C 180,E1 -13133.343,E2 -13133.343} C_VEL
LIN {X 0,Y 363.39,Z 433.797,A -85,B 0,C 180,E1 -13134.451,E2 -13134.451} C_VEL
LIN {X 0,Y 363.13,Z 434.821,A -85,B 0,C 180,E1 -13135.56,E2 -13135.56} C_VEL
LIN {X 0,Y 362.801,Z 435.461,A -85,B 0,C 180,E1 -13136.669,E2 -13136.669} C_VEL
LIN {X 0,Y 362.587,Z 435.683,A -85,B 0,C 180,E1 -13137.778,E2 -13137.778} C_VEL
LIN {X 0,Y 362.302,Z 435.495,A -85,B 0,C 180,E1 -13138.889,E2 -13138.889} C_VEL
LIN {X 0,Y 362.08,Z 434.843,A -85,B 0,C 180,E1 -13140,E2 -13140} C_VEL
LIN {X 0,Y 362.092,Z 433.759,A -85,B 0,C 180,E1 -13141.112,E2 -13141.112} C_VEL
LIN {X 0,Y 362.022,Z 432.281,A -85,B 0,C 180,E1 -13142.225,E2 -13142.225} C_VEL
LIN {X 0,Y 361.972,Z 429.206,A -85,B 0,C 180,E1 -13143.897,E2 -13143.897} C_VEL
LIN {X 0,Y 362.173,Z 425.067,A -85,B 0,C 180,E1 -13145.568,E2 -13145.568} C_VEL
LIN {X 0,Y 362.504,Z 418.786,A -85,B 0,C 180,E1 -13147.52,E2 -13147.52} C_VEL
LIN {X 0,Y 362.867,Z 410.679,A -85,B 0,C 180,E1 -13149.476,E2 -13149.476} C_VEL
LIN {X 0,Y 363.415,Z 402.01,A -85,B 0,C 180,E1 -13151.151,E2 -13151.151} C_VEL
LIN {X 0,Y 364.058,Z 391.284,A -85,B 0,C 180,E1 -13152.827,E2 -13152.827} C_VEL
LIN {X 0,Y 364.704,Z 380.315,A -85,B 0,C 180,E1 -13154.223,E2 -13154.223} C_VEL
LIN {X 0,Y 365.415,Z 368.129,A -85,B 0,C 180,E1 -13155.477,E2 -13155.477} C_VEL
LIN {X 0,Y 365.92,Z 355.797,A -85,B 0,C 180,E1 -13156.507,E2 -13156.507} C_VEL
LIN {X 0,Y 366.463,Z 342.516,A -85,B 0,C 180,E1 -13157.365,E2 -13157.365} C_VEL
LIN {X 0,Y 366.855,Z 328.805,A -85,B 0,C 180,E1 -13158.03,E2 -13158.03} C_VEL
LIN {X 0,Y 367.268,Z 313.922,A -85,B 0,C 180,E1 -13158.514,E2 -13158.514} C_VEL
LIN {X 0,Y 369.73,Z 225.372,A -85,B 0,C 180,E1 -13160.873,E2 -13160.873} C_VEL
LIN {X 0,Y 366.132,Z 202.768,A -85,B 0,C 180,E1 -13161.685,E2 -13161.685} C_VEL
LIN {X 0,Y 367.593,Z 185.358,A -85,B 0,C 180,E1 -13165.161,E2 -13165.161} C_VEL
LIN {X 0,Y 367.411,Z 181.572,A -85,B 0,C 180,E1 -13165.966,E2 -13165.966} C_VEL
LIN {X 0,Y 364.357,Z 167.735,A -85,B 0,C 180,E1 -13169.102,E2 -13169.102} C_VEL
LIN {X 0,Y 361.91,Z 157.031,A -85,B 0,C 180,E1 -13171.622,E2 -13171.622} C_VEL
LIN {X 0,Y 361.873,Z 157.034,A -85,B 0,C 180,E1 -13175.636,E2 -13175.636} C_VEL
LIN {X 0,Y 361.836,Z 157.032,A -85,B 0,C 180,E1 -13179.018,E2 -13179.018} C_VEL
LIN {X 0,Y 361.839,Z 157.035,A -85,B 0,C 180,E1 -13182.829,E2 -13182.829} C_VEL
LIN {X 0,Y 361.84,Z 157.037,A -85,B 0,C 180,E1 -13185.943,E2 -13185.943} C_VEL
LIN {X 0,Y 361.841,Z 157.036,A -85,B 0,C 180,E1 -13189.244,E2 -13189.244} C_VEL
LIN {X 0,Y 361.868,Z 157.033,A -85,B 0,C 180,E1 -13192.777,E2 -13192.777} C_VEL
LIN {X 0,Y 361.877,Z 157.051,A -85,B 0,C 180,E1 -13195.721,E2 -13195.721} C_VEL
LIN {X 0,Y 366.644,Z 171.124,A -85,B 0,C 180,E1 -13198.357,E2 -13198.357} C_VEL
LIN {X 0,Y 375.859,Z 189.539,A -85,B 0,C 180,E1 -13199.651,E2 -13199.651} C_VEL
LIN {X 0,Y 380.929,Z 200.988,A -85,B 0,C 180,E1 -13200.351,E2 -13200.351} C_VEL
LIN {X 0,Y 378.921,Z 284.505,A -85,B 0,C 180,E1 -13201.961,E2 -13201.961} C_VEL
LIN {X 0,Y 377.534,Z 338.148,A -85,B 0,C 180,E1 -13203.014,E2 -13203.014} C_VEL
LIN {X 0,Y 376.975,Z 352.753,A -85,B 0,C 180,E1 -13203.492,E2 -13203.492} C_VEL
LIN {X 0,Y 376.205,Z 365.205,A -85,B 0,C 180,E1 -13204.056,E2 -13204.056} C_VEL
LIN {X 0,Y 375.116,Z 379.544,A -85,B 0,C 180,E1 -13204.918,E2 -13204.918} C_VEL
LIN {X 0,Y 373.691,Z 393.651,A -85,B 0,C 180,E1 -13206.001,E2 -13206.001} C_VEL
LIN {X 0,Y 372.075,Z 406.486,A -85,B 0,C 180,E1 -13207.217,E2 -13207.217} C_VEL
LIN {X 0,Y 370.335,Z 419.095,A -85,B 0,C 180,E1 -13208.683,E2 -13208.683} C_VEL
LIN {X 0,Y 368.83,Z 430.082,A -85,B 0,C 180,E1 -13210.23,E2 -13210.23} C_VEL
LIN {X 0,Y 367.225,Z 439.967,A -85,B 0,C 180,E1 -13211.88,E2 -13211.88} C_VEL
LIN {X 0,Y 365.554,Z 449.862,A -85,B 0,C 180,E1 -13213.869,E2 -13213.869} C_VEL
LIN {X 0,Y 364.178,Z 458.617,A -85,B 0,C 180,E1 -13216.04,E2 -13216.04} C_VEL
LIN {X 0,Y 362.969,Z 465.874,A -85,B 0,C 180,E1 -13218.268,E2 -13218.268} C_VEL
LIN {X 0,Y 362.154,Z 471.614,A -85,B 0,C 180,E1 -13220.504,E2 -13220.504} C_VEL
LIN {X 0,Y 361.579,Z 475.68,A -85,B 0,C 180,E1 -13222.574,E2 -13222.574} C_VEL
LIN {X 0,Y 361.246,Z 478.45,A -85,B 0,C 180,E1 -13224.416,E2 -13224.416} C_VEL
LIN {X 0,Y 361.046,Z 480.718,A -85,B 0,C 180,E1 -13226.651,E2 -13226.651} C_VEL
LIN {X 0,Y 360.948,Z 481.182,A -85,B 0,C 180,E1 -13227.37,E2 -13227.37} C_VEL
LIN {X 0,Y 360.214,Z 481.75,A -85,B 0,C 180,E1 -13228.297,E2 -13228.297} C_VEL
LIN {X 0,Y 357.305,Z 482.404,A -85,B 0,C 180,E1 -13229.808,E2 -13229.808} C_VEL
LIN {X 0,Y 354.905,Z 482.5,A -85,B 0,C 180,E1 -13231.031,E2 -13231.031} C_VEL
LIN {X 0,Y 353.912,Z 482.223,A -85,B 0,C 180,E1 -13231.976,E2 -13231.976} C_VEL
LIN {X 0,Y 353.85,Z 482.051,A -85,B 0,C 180,E1 -13232.295,E2 -13232.295} C_VEL
LIN {X 0,Y 354.146,Z 480.401,A -85,B 0,C 180,E1 -13234.551,E2 -13234.551} C_VEL
LIN {X 0,Y 354.353,Z 477.624,A -85,B 0,C 180,E1 -13236.833,E2 -13236.833} C_VEL
LIN {X 0,Y 354.983,Z 473.62,A -85,B 0,C 180,E1 -13239.112,E2 -13239.112} C_VEL
LIN {X 0,Y 355.775,Z 468.301,A -85,B 0,C 180,E1 -13241.392,E2 -13241.392} C_VEL
LIN {X 0,Y 356.852,Z 461.51,A -85,B 0,C 180,E1 -13243.669,E2 -13243.669} C_VEL
LIN {X 0,Y 358.174,Z 453.78,A -85,B 0,C 180,E1 -13245.759,E2 -13245.759} C_VEL
LIN {X 0,Y 359.667,Z 445.417,A -85,B 0,C 180,E1 -13247.629,E2 -13247.629} C_VEL
LIN {X 0,Y 361.505,Z 434.75,A -85,B 0,C 180,E1 -13249.592,E2 -13249.592} C_VEL
LIN {X 0,Y 363.187,Z 423.788,A -85,B 0,C 180,E1 -13251.272,E2 -13251.272} C_VEL
LIN {X 0,Y 364.999,Z 411.722,A -85,B 0,C 180,E1 -13252.797,E2 -13252.797} C_VEL
LIN {X 0,Y 366.818,Z 398.377,A -85,B 0,C 180,E1 -13254.174,E2 -13254.174} C_VEL
LIN {X 0,Y 368.28,Z 385.303,A -85,B 0,C 180,E1 -13255.275,E2 -13255.275} C_VEL
LIN {X 0,Y 369.584,Z 371.368,A -85,B 0,C 180,E1 -13256.208,E2 -13256.208} C_VEL
LIN {X 0,Y 370.507,Z 356.754,A -85,B 0,C 180,E1 -13256.962,E2 -13256.962} C_VEL
LIN {X 0,Y 371.2,Z 342.46,A -85,B 0,C 180,E1 -13257.482,E2 -13257.482} C_VEL
LIN {X 0,Y 371.718,Z 322.104,A -85,B 0,C 180,E1 -13257.937,E2 -13257.937} C_VEL
LIN {X 0,Y 374.877,Z 203.721,A -85,B 0,C 180,E1 -13260.235,E2 -13260.235} C_VEL
LIN {X 0,Y 371.448,Z 195.351,A -85,B 0,C 180,E1 -13260.735,E2 -13260.735} C_VEL
LIN {X 0,Y 361.38,Z 175.051,A -85,B 0,C 180,E1 -13262.175,E2 -13262.175} C_VEL
LIN {X 0,Y 359.549,Z 171.489,A -85,B 0,C 180,E1 -13262.488,E2 -13262.488} C_VEL
LIN {X 0,Y 354.846,Z 157.909,A -85,B 0,C 180,E1 -13265.093,E2 -13265.093} C_VEL
LIN {X 0,Y 354.803,Z 157.915,A -85,B 0,C 180,E1 -13267.881,E2 -13267.881} C_VEL
LIN {X 0,Y 354.784,Z 157.897,A -85,B 0,C 180,E1 -13271.171,E2 -13271.171} C_VEL
LIN {X 0,Y 354.762,Z 157.911,A -85,B 0,C 180,E1 -13274.506,E2 -13274.506} C_VEL
LIN {X 0,Y 354.805,Z 157.907,A -85,B 0,C 180,E1 -13277.664,E2 -13277.664} C_VEL
LIN {X 0,Y 354.829,Z 157.904,A -85,B 0,C 180,E1 -13280.668,E2 -13280.668} C_VEL
LIN {X 0,Y 354.814,Z 157.91,A -85,B 0,C 180,E1 -13284.299,E2 -13284.299} C_VEL
LIN {X 0,Y 354.79,Z 157.916,A -85,B 0,C 180,E1 -13287.667,E2 -13287.667} C_VEL
LIN {X 0,Y 354.86,Z 157.892,A -85,B 0,C 180,E1 -13290.62,E2 -13290.62} C_VEL
LIN {X 0,Y 354.889,Z 157.896,A -85,B 0,C 180,E1 -13294.172,E2 -13294.172} C_VEL
LIN {X 0,Y 354.82,Z 157.911,A -85,B 0,C 180,E1 -13297.893,E2 -13297.893} C_VEL
LIN {X 0,Y 354.912,Z 157.889,A -85,B 0,C 180,E1 -13301.891,E2 -13301.891} C_VEL
LIN {X 0,Y 354.932,Z 157.888,A -85,B 0,C 180,E1 -13305.98,E2 -13305.98} C_VEL
LIN {X 0,Y 354.967,Z 157.892,A -85,B 0,C 180,E1 -13309.735,E2 -13309.735} C_VEL
LIN {X 0,Y 355.103,Z 157.87,A -85,B 0,C 180,E1 -13312.036,E2 -13312.036} C_VEL
LIN {X 0,Y 355.082,Z 157.861,A -85,B 0,C 180,E1 -13314.32,E2 -13314.32} C_VEL
LIN {X 0,Y 355.235,Z 157.857,A -85,B 0,C 180,E1 -13317.732,E2 -13317.732} C_VEL
LIN {X 0,Y 355.388,Z 157.82,A -85,B 0,C 180,E1 -13320,E2 -13320} C_VEL
LIN {X 0,Y 355.235,Z 157.853,A -85,B 0,C 180,E1 -13322.268,E2 -13322.268} C_VEL
LIN {X 0,Y 355.127,Z 157.852,A -85,B 0,C 180,E1 -13326.819,E2 -13326.819} C_VEL
LIN {X 0,Y 355.004,Z 157.885,A -85,B 0,C 180,E1 -13329.112,E2 -13329.112} C_VEL
LIN {X 0,Y 354.91,Z 157.879,A -85,B 0,C 180,E1 -13332.581,E2 -13332.581} C_VEL
LIN {X 0,Y 354.881,Z 157.901,A -85,B 0,C 180,E1 -13336.096,E2 -13336.096} C_VEL
LIN {X 0,Y 354.89,Z 157.885,A -85,B 0,C 180,E1 -13338.473,E2 -13338.473} C_VEL
LIN {X 0,Y 354.824,Z 157.911,A -85,B 0,C 180,E1 -13342.107,E2 -13342.107} C_VEL
LIN {X 0,Y 354.888,Z 157.895,A -85,B 0,C 180,E1 -13345.828,E2 -13345.828} C_VEL
LIN {X 0,Y 354.807,Z 157.899,A -85,B 0,C 180,E1 -13349.683,E2 -13349.683} C_VEL
LIN {X 0,Y 354.796,Z 157.907,A -85,B 0,C 180,E1 -13353.703,E2 -13353.703} C_VEL
LIN {X 0,Y 354.792,Z 157.917,A -85,B 0,C 180,E1 -13356.46,E2 -13356.46} C_VEL
LIN {X 0,Y 354.815,Z 157.876,A -85,B 0,C 180,E1 -13359.425,E2 -13359.425} C_VEL
LIN {X 0,Y 354.782,Z 157.91,A -85,B 0,C 180,E1 -13362.869,E2 -13362.869} C_VEL
LIN {X 0,Y 354.844,Z 157.91,A -85,B 0,C 180,E1 -13366.118,E2 -13366.118} C_VEL
LIN {X 0,Y 354.858,Z 157.932,A -85,B 0,C 180,E1 -13369.191,E2 -13369.191} C_VEL
LIN {X 0,Y 361.007,Z 178.813,A -85,B 0,C 180,E1 -13372.956,E2 -13372.956} C_VEL
LIN {X 0,Y 366.044,Z 196.273,A -85,B 0,C 180,E1 -13375.905,E2 -13375.905} C_VEL
LIN {X 0,Y 367.092,Z 200.654,A -85,B 0,C 180,E1 -13376.606,E2 -13376.606} C_VEL
LIN {X 0,Y 365.738,Z 211.406,A -85,B 0,C 180,E1 -13378.041,E2 -13378.041} C_VEL
LIN {X 0,Y 366.368,Z 219.775,A -85,B 0,C 180,E1 -13378.45,E2 -13378.45} C_VEL
LIN {X 0,Y 372.112,Z 268.539,A -85,B 0,C 180,E1 -13380.044,E2 -13380.044} C_VEL
LIN {X 0,Y 372.587,Z 274.818,A -85,B 0,C 180,E1 -13380.221,E2 -13380.221} C_VEL
LIN {X 0,Y 369.5,Z 393.43,A -85,B 0,C 180,E1 -13382.535,E2 -13382.535} C_VEL
LIN {X 0,Y 368.623,Z 408.483,A -85,B 0,C 180,E1 -13383.001,E2 -13383.001} C_VEL
LIN {X 0,Y 367.272,Z 423.215,A -85,B 0,C 180,E1 -13383.661,E2 -13383.661} C_VEL
LIN {X 0,Y 365.798,Z 436.406,A -85,B 0,C 180,E1 -13384.45,E2 -13384.45} C_VEL
LIN {X 0,Y 364.178,Z 449.982,A -85,B 0,C 180,E1 -13385.488,E2 -13385.488} C_VEL
LIN {X 0,Y 362.173,Z 463.057,A -85,B 0,C 180,E1 -13386.712,E2 -13386.712} C_VEL
LIN {X 0,Y 360.434,Z 475.143,A -85,B 0,C 180,E1 -13388.106,E2 -13388.106} C_VEL
LIN {X 0,Y 358.72,Z 486.331,A -85,B 0,C 180,E1 -13389.652,E2 -13389.652} C_VEL
LIN {X 0,Y 357.254,Z 496.653,A -85,B 0,C 180,E1 -13391.358,E2 -13391.358} C_VEL
LIN {X 0,Y 355.769,Z 506.739,A -85,B 0,C 180,E1 -13393.357,E2 -13393.357} C_VEL
LIN {X 0,Y 354.775,Z 515.136,A -85,B 0,C 180,E1 -13395.372,E2 -13395.372} C_VEL
LIN {X 0,Y 354.041,Z 522.1,A -85,B 0,C 180,E1 -13397.389,E2 -13397.389} C_VEL
LIN {X 0,Y 353.602,Z 528.576,A -85,B 0,C 180,E1 -13399.697,E2 -13399.697} C_VEL
LIN {X 0,Y 353.536,Z 533.6,A -85,B 0,C 180,E1 -13402.003,E2 -13402.003} C_VEL
LIN {X 0,Y 353.637,Z 537.288,A -85,B 0,C 180,E1 -13404.299,E2 -13404.299} C_VEL
